(* CoDeSys 2.3.9.48 project: Code_def.pro *)
(* Libraries: standard.lib 2.6.14 10:37:46, Iecsfc.lib 2.6.14 10:37:46, Util.lib 15.3.18 01:28:42, SysLibTime.lib 25.6.18 19:33:14, SysTaskInfo.lib 25.6.18 19:33:14, Syslibs\SysLibRtc.lib 25.6.18 19:33:14, SysLibMem.lib 25.6.18 19:33:14, SYSLIBCALLBACK.LIB 25.6.18 19:33:14, BusDiag.LIB 25.6.18 19:33:14, SysExt_AC500_V10.lib 25.6.18 19:33:14, SysInt_AC500_V10.LIB 25.6.18 19:33:14, MODBUS_AC500_V10.lib 25.6.18 19:33:14 *)

(* PLC configuration (modules and I/O channels)
CPU parameters [AC500_CPU] node 0, in %IB0 out %QB0 {AutoRunType = On; ErrLEDType = On; CheckBatteryType = Off; OutputsInStopType = Off in hardware and online; StopErrorClassType = E2; WarmstartOnFK2Type = Off; FloatingPointExceptionType = E2 failure; IOSimulationModeType = Off; NumberRetainSegmentsType = 8; StartRetainM0Type = 0; EndRetainM0Type = 0; StartRetainM1Type = 0; EndRetainM1Type = 0; StartRetainM2Type = 0; EndRetainM2Type = 0; StartRetainM3Type = 0; EndRetainM3Type = 0; StartRetainM4Type = 0; EndRetainM4Type = 0; StartRetainM5Type = 0; EndRetainM5Type = 0; StartRetainM6Type = 0; EndRetainM6Type = 0; StartRetainM7Type = 0; EndRetainM7Type = 0}
AT %IW0 [WordInputNoSpace] Input 0-15
AT %IB0 [ByteInputNoSpace] Input 0-7
CabStop AT %IX0.0 [BoolInput] Input 0
CabCallP3 AT %IX0.1 [BoolInput] Input 1
CabCallP2 AT %IX0.2 [BoolInput] Input 2
CabCallP1 AT %IX0.3 [BoolInput] Input 3
CabCallP0 AT %IX0.4 [BoolInput] Input 4
CabObstacle AT %IX0.5 [BoolInput] Input 5
Floor3DwBt AT %IX0.6 [BoolInput] Input 6
Floor3DoorClosed AT %IX0.7 [BoolInput] Input 7
AT %IB1 [ByteInputNoSpace] Input 8-15
Floor3DoorOpened AT %IX1.0 [BoolInput] Input 8
Floor3CabPresence AT %IX1.1 [BoolInput] Input 9
Floor2UpBt AT %IX1.2 [BoolInput] Input 10
Floor2DwBt AT %IX1.3 [BoolInput] Input 11
Floor2DoorClosed AT %IX1.4 [BoolInput] Input 12
Floor2DoorOpened AT %IX1.5 [BoolInput] Input 13
Floor2CabPresence AT %IX1.6 [BoolInput] Input 14
Floor1UpBt AT %IX1.7 [BoolInput] Input 15
AT %IW1 [WordInputNoSpace] Input 16-31
AT %IB2 [ByteInputNoSpace] Input 16-23
AT %IX2.0 [BoolInput] Input 16
AT %IX2.1 [BoolInput] Input 17
AT %IX2.2 [BoolInput] Input 18
AT %IX2.3 [BoolInput] Input 19
AT %IX2.4 [BoolInput] Input 20
AT %IX2.5 [BoolInput] Input 21
AT %IX2.6 [BoolInput] Input 22
AT %IX2.7 [BoolInput] Input 23
AT %IB3 [ByteInputNoSpace] Input 24-31
AT %IX3.0 [BoolInput] Input 24
AT %IX3.1 [BoolInput] Input 25
AT %IX3.2 [BoolInput] Input 26
AT %IX3.3 [BoolInput] Input 27
AT %IX3.4 [BoolInput] Input 28
AT %IX3.5 [BoolInput] Input 29
AT %IX3.6 [BoolInput] Input 30
AT %IX3.7 [BoolInput] Input 31
AT %QW0 [WordOutputNoSpace] Output 16-31
AT %QB0 [ByteOutputNoSpace] Output 16-23
CabGoUp AT %QX0.0 [BoolOutput] Output 16
CabGoDown AT %QX0.1 [BoolOutput] Output 17
CabLight AT %QX0.2 [BoolOutput] Output 18
CabLed3 AT %QX0.3 [BoolOutput] Output 19
CabLed2 AT %QX0.4 [BoolOutput] Output 20
CabLed1 AT %QX0.5 [BoolOutput] Output 21
Floor3LedDw AT %QX0.6 [BoolOutput] Output 22
CabLed0 AT %QX0.7 [BoolOutput] Output 23
AT %QB1 [ByteOutputNoSpace] Output 24-31
Floor3DoorClose AT %QX1.0 [BoolOutput] Output 24
Floor3DoorOpen AT %QX1.1 [BoolOutput] Output 25
Floor2LedUp AT %QX1.2 [BoolOutput] Output 26
Floor2LedDw AT %QX1.3 [BoolOutput] Output 27
Floor2DoorClose AT %QX1.4 [BoolOutput] Output 28
Floor2DoorOpen AT %QX1.5 [BoolOutput] Output 29
Floor1LedDw AT %QX1.6 [BoolOutput] Output 30
Floor1LedUp AT %QX1.7 [BoolOutput] Output 31
Fast counter [Module_2FastCounter] node 3, in %IB4 out %QB2
  AT %ID1 [DWordInput] Istwert/Actual value 1
  AT %ID2 [DWordInput] Istwert/Actual value 2
  AT %IB12 [ByteInputNoBits] Statusbyte/State byte 1
  AT %IB13 [ByteInputNoBits] Statusbyte/State byte 2
  AT %QD1 [DWordOutput] Startwert/Start value 1
  AT %QD2 [DWordOutput] Endwert/End value 1
  AT %QD3 [DWordOutput] Startwert/Start value 2
  AT %QD4 [DWordOutput] Endwert/End value 2
  AT %QB20 [ByteOutputNoBits] Steuerbyte/Control byte 1
  AT %QB21 [ByteOutputNoBits] Steuerbyte/Control byte 2
AT %IW7 [WordInputNoSpace] Input 0-15
AT %IB14 [ByteInputNoSpace] Input 0-7
Floor1DwBt AT %IX14.0 [BoolInput] Input 0
Floor1DoorClosed AT %IX14.1 [BoolInput] Input 1
Floor1DoorOpened AT %IX14.2 [BoolInput] Input 2
Floor1CabPresence AT %IX14.3 [BoolInput] Input 3
Floor0UpBt AT %IX14.4 [BoolInput] Input 4
Floor0DoorClosed AT %IX14.5 [BoolInput] Input 5
Floor0DoorOpened AT %IX14.6 [BoolInput] Input 6
Floor0CabPresence AT %IX14.7 [BoolInput] Input 7
AT %IB15 [ByteInputNoSpace] Input 8-15
AT %IX15.0 [BoolInput] Input 8
AT %IX15.1 [BoolInput] Input 9
AT %IX15.2 [BoolInput] Input 10
AT %IX15.3 [BoolInput] Input 11
AT %IX15.4 [BoolInput] Input 12
AT %IX15.5 [BoolInput] Input 13
AT %IX15.6 [BoolInput] Input 14
AT %IX15.7 [BoolInput] Input 15
AT %IW8 [WordInputNoSpace] Input 16-31
AT %IB16 [ByteInputNoSpace] Input 16-23
AT %IX16.0 [BoolInput] Input 16
AT %IX16.1 [BoolInput] Input 17
AT %IX16.2 [BoolInput] Input 18
AT %IX16.3 [BoolInput] Input 19
AT %IX16.4 [BoolInput] Input 20
AT %IX16.5 [BoolInput] Input 21
AT %IX16.6 [BoolInput] Input 22
AT %IX16.7 [BoolInput] Input 23
AT %IB17 [ByteInputNoSpace] Input 24-31
AT %IX17.0 [BoolInput] Input 24
AT %IX17.1 [BoolInput] Input 25
AT %IX17.2 [BoolInput] Input 26
AT %IX17.3 [BoolInput] Input 27
AT %IX17.4 [BoolInput] Input 28
AT %IX17.5 [BoolInput] Input 29
AT %IX17.6 [BoolInput] Input 30
AT %IX17.7 [BoolInput] Input 31
AT %QW11 [WordOutputNoSpace] Output 16-31
AT %QB22 [ByteOutputNoSpace] Output 16-23
Floor1DoorClose AT %QX22.0 [BoolOutput] Output 16
Floor1DoorOpen AT %QX22.1 [BoolOutput] Output 17
Floor0LedUp AT %QX22.2 [BoolOutput] Output 18
Floor0DoorClose AT %QX22.3 [BoolOutput] Output 19
Floor0DoorOpen AT %QX22.4 [BoolOutput] Output 20
AT %QX22.5 [BoolOutput] Output 21
AT %QX22.6 [BoolOutput] Output 22
AT %QX22.7 [BoolOutput] Output 23
AT %QB23 [ByteOutputNoSpace] Output 24-31
AT %QX23.0 [BoolOutput] Output 24
AT %QX23.1 [BoolOutput] Output 25
AT %QX23.2 [BoolOutput] Output 26
AT %QX23.3 [BoolOutput] Output 27
AT %QX23.4 [BoolOutput] Output 28
AT %QX23.5 [BoolOutput] Output 29
AT %QX23.6 [BoolOutput] Output 30
AT %QX23.7 [BoolOutput] Output 31
Fast counter [Module_2FastCounter] node 3, in %IB18 out %QB24
  AT %ID5 [DWordInput] Istwert/Actual value 1
  AT %ID6 [DWordInput] Istwert/Actual value 2
  AT %IB28 [ByteInputNoBits] Statusbyte/State byte 1
  AT %IB29 [ByteInputNoBits] Statusbyte/State byte 2
  AT %QD6 [DWordOutput] Startwert/Start value 1
  AT %QD7 [DWordOutput] Endwert/End value 1
  AT %QD8 [DWordOutput] Startwert/Start value 2
  AT %QD9 [DWordOutput] Endwert/End value 2
  AT %QB40 [ByteOutputNoBits] Steuerbyte/Control byte 1
  AT %QB41 [ByteOutputNoBits] Steuerbyte/Control byte 2
COM1 - MODBUS [AC500_COM1_MODBUS] node 0, in %IB1000 out %QB1000 {COMEnableLoginType = Disabled; COMRTSctrlType = telegram; COMTLSType = 0; COMCDLYType = 0; COMCharTimeoutType = 0; COMTelEndSelType = character timeout; COMTelEndValCharType = 16#00; COMTelEndValWertType = 3; COMChecksumType = CRC16; COMHandshakeType = none; COMBaudType = 19200; COMParityType = none; COMDataBitType = 8; COMStopBitType = 1; COMOperatingModeType = Slave; COMAdressType = 1; COMDisableWriteStartSeg0Type = 0; COMDisableWriteEndSeg0Type = 0; COMDisableReadStartSeg0Type = 0; COMDisableReadEndSeg0Type = 0; COMDisableWriteStartSeg1Type = 0; COMDisableWriteEndSeg1Type = 0; COMDisableReadStartSeg1Type = 0; COMDisableReadEndSeg1Type = 0}
COM2 - Online access [AC500_COM2_Programming] node 1, in %IB2000 out %QB2000 {COMEnableLoginType = Disabled; COMRTSctrlType = telegram; COMTLSType = 0; COMCDLYType = 0; COMCharTimeoutType = 0; COMTelEndSelType = none; COMTelEndValCharType = 16#00; COMTelEndValWertType = 0; COMChecksumType = none; COMHandshakeType = none; COMBaudType = 19200; COMParityType = none; COMDataBitType = 8; COMStopBitType = 1}
FBP - none [AC500_FBP_None] node 2, in %IB3000 out %QB3000
Couplers [AC500_Int_Empty] node 3, in %IB0.0 out %QB0.0
  Internal - none [AC500_IntEmpty] node 0, in %IB4096 out %QB4096 {RunConfigFaultType = No; MaxWaitRunType = 3000; MinUpdateTimeType = 10; ReserveWord0Type = 0; ReserveWord1Type = 0; ReserveWord2Type = 0}
*)

(* Task configuration *)
TASK NewTask (PRIORITY := 10, INTERVAL := T#1ms);
	Main();
END_TASK

(* Global variable list: Global_Variables *)
VAR_GLOBAL
	N: INT:= 6;						(*==============================================================*)
	CabCall: ARRAY [0..5] OF INT;  (*==============================================================*)
	Cabin: CabinDef;
	CallFloor0: BOOL := FALSE;
	CallFloor1: BOOL := FALSE;
	CallFloor2: BOOL := FALSE;
	CallFloor3: BOOL := FALSE;
	Close0 AT %MX0.1.5: BOOL :=FALSE;
	Close1 AT %MX0.1.6: BOOL :=FALSE;
	Close2 AT %MX0.1.7: BOOL :=FALSE;
	Close3 AT %MX0.1.0: BOOL :=FALSE;
	CurrentFloor: UINT;
	DesiredFloor AT %MW0.50: INT;
	Displacement: INT := 450;
	Door0:	INT :=0;
	Door1: INT :=0;
	Door2: INT :=0;
	Door3: INT :=0;
	Door : ARRAY [0..5] OF INT;		(*==============================================================*)
	DoorClosed0 AT %MX0.6.0: BOOL;
	DoorClosed1 AT %MX0.6.2: BOOL;
	DoorClosed2 AT %MX0.6.4: BOOL;
	DoorClosed3 AT %MX0.6.6: BOOL;
	DoorOpened0 AT %MX0.6.1: BOOL;
	DoorOpened1 AT %MX0.6.3: BOOL;
	DoorOpened2 AT %MX0.6.5: BOOL;
	DoorOpened3 AT %MX0.6.7: BOOL;
	DwCall: ARRAY [0..5] OF INT;		(*==============================================================*)
	DwCall1 AT %MW0.61: INT;
	DwCall2 AT %MW0.62: INT;
	DwCall3 AT %MW0.63: INT;
	DwCall4 AT %MW0.64: INT;
	EndMovement: BOOL;
	EndMovementObstacle: BOOL := FALSE;
	EndOpening: BOOL;
	EndOpeningObstacle: BOOL := FALSE;
	Error AT %MW0.4: INT := 0;
	ErrorOpeningDoor: ARRAY [0..5] OF BOOL;	(*==============================================================*)
	ErrorClosingDoor: ARRAY [0..5] OF BOOL;(*==============================================================*)
	Floor: ARRAY[0..5] OF FloorDef;  			(*==============================================================*)
	FloorIndicator AT %MW0.2: UINT;
	GoDw AT %MX0.0.3: BOOL :=FALSE;
	GoUp AT %MX0.0.2: BOOL :=FALSE;
	Init AT %MX0.0.0: BOOL := FALSE;
	IntCall1 AT %MW0.53: INT;
	IntCall2 AT %MW0.54: INT;
	IntCall3 AT %MW0.55: INT;
	IntCall4 AT %MW0.56: INT;

	IntermittingLightOFF: BOOL;
	IntermittingLightON: BOOL;
	isBetween: ARRAY [0..5] OF BOOL;  (*==============================================================*)
	LimitWeight AT %MW0.52: INT:=320;
	Man AT %MX0.0.1:  BOOL := FALSE;

	MovedDw: BOOL;
	MovedUp: BOOL;
	MovingDw: BOOL;
	MovingUp: BOOL;
	Multiple: BOOL := FALSE;
	ObstacleCase: BOOL := FALSE;
	ObstacleOccurred: BOOL := FALSE;
	Open0 AT %MX0.1.1: BOOL := FALSE;
	Open1 AT %MX0.1.2: BOOL := FALSE;
	Open2 AT %MX0.1.3: BOOL := FALSE;
	Open3 AT %MX0.1.4: BOOL := FALSE;
	Optimized: BOOL := FALSE;
	PreviousLogic: INT;
	Queue: ARRAY [0..5] OF INT;			(*==============================================================*)
	Queue1 AT %MW0.65: INT;
	Queue2 AT %MW0.66: INT;
	Queue3 AT %MW0.67: INT;
	Queue4 AT %MW0.68: INT;
	ReadyToDelete: BOOL;
	ReadyToMove: BOOL;
	Single: BOOL := FALSE;
	StartClose: BOOL;
	StartCloseAfterObstacle: BOOL;
	StopOccurred: BOOL := FALSE;
	TimerCabLightOFF: BOOL;
	TimerDelete: BOOL;
	TimerDoor: BOOL;
	TimerDoorAfterObstacle: BOOL;
	TimerErrorCabin: BOOL := FALSE;
	TimerErrorOpeningDoor: ARRAY [0..5] OF BOOL:= FALSE; (*==============================================================*)
	TimerErrorClosingDoor: ARRAY [0..5] OF BOOL:= FALSE;(*==============================================================*)
	TimerIntermittingLightOFF: BOOL;
	TimerIntermittingLightON: BOOL;
	TimerReOpening: BOOL;
	UpCall: ARRAY [0..5] OF INT;(*==============================================================*)
	UpCall1 AT %MW0.57: INT;
	UpCall2 AT %MW0.58: INT;
	UpCall3 AT %MW0.59: INT;
	UpCall4 AT %MW0.60: INT;
	Weight AT %MW0.51: INT;
END_VAR

(* Data type *)
TYPE CabinDef :
STRUCT

	Call:ARRAY [0..5] OF BOOL;	(*==============================================================*)
	GoUp: BOOL;
	GoDown: BOOL;
	Light: BOOL;
	Obstacle: BOOL;
	Stop: BOOL;
	ErrorCabin: BOOL;

END_STRUCT
END_TYPE

(* Data type *)
TYPE FloorDef :
STRUCT

	DoorClose: BOOL;
	DoorOpen: BOOL;
	DoorOpened: BOOL;
	DoorClosed: BOOL;
	CabPresence: BOOL;
	CallUp: BOOL;
	CallDw: BOOL;
	CabLed: BOOL;
	LedUp: BOOL;
	LedDw: BOOL;

END_STRUCT
END_TYPE

(* POU Main, ST *)
PROGRAM Main
VAR
	CabLightOFF: BOOL;
	i: INT;
	Logic AT %MW0.5: INT := 3;
	OverWeight: BOOL;
	Sim: BOOL := FALSE;
	TimerStop: BOOL;
	TON_CabLightOFF: TON;
	TON_Delete: TON;
	TON_Door: TON;
	TON_ErrorCabin: TON;
	TON_ErrorOpeningDoor: ARRAY[0..5] OF TON;   (*==============================================================*)
	TON_ErrorClosingDoor: ARRAY[0..5] OF TON;	(*==============================================================*)
	TON_Obstacle: TON;
	TON_ReOpening: TON;
	TON_StopLightOFF: TON;
	TON_StopLightON: TON;
	CountDoorClosed: INT;
	CountErrorClosingDoor : INT;
	CountErrorOpeningDoor: INT;
END_VAR
IF (Sim = FALSE) THEN
	ASS_INPUT;
	(*HMI;*)
ELSE
	SIMULATION_INPUT;
END_IF

IF (Man = TRUE) THEN
	(*MANUAL;*)
	;
ELSE

(*-------------------------------------------------------initialization----------------------------------------------------*)
	IF( Init = FALSE) THEN
		Init := Initialize();
	ELSE

		TON_StopLightOFF(IN:= TimerIntermittingLightOFF, PT:= T#1s, Q=> IntermittingLightOFF);
		TON_StopLightON(IN:= TimerIntermittingLightON, PT:= T#1s, Q=> IntermittingLightON);

		(*CountDoorClosed = N if all doors are closed 		    *)
		(*					   < N if at least one door is opened *)
		(*CountErrorClosingDoor = N if no error during closing door*)
		(*							 <N ia there is an error during closing door*)
		(*CountErrorOpeningDoor = N if no error during opening door*)
		(*							 <N ia there is an error during opening door*)
		CountDoorClosed := 0;
		CountErrorClosingDoor := 0;
		CountErrorOpeningDoor  := 0;

		FOR i := 0 TO N-1 DO
			IF (Floor[i].DoorClosed = TRUE) THEN
				CountDoorClosed := CountDoorClosed +1;
			END_IF
			IF (ErrorClosingDoor[i] = FALSE) THEN
				CountErrorClosingDoor := CountErrorClosingDoor + 1;
			END_IF
			IF (ErrorOpeningDoor[i] = FALSE) THEN
				CountErrorOpeningDoor := CountErrorOpeningDoor + 1;
			END_IF
		END_FOR


		IF (CountDoorClosed < N AND Weight > LimitWeight) THEN
			OverWeight := TRUE;
		ELSE
			OverWeight:= FALSE;
		END_IF

		IF (Cabin.ErrorCabin = FALSE AND CountErrorClosingDoor = N AND CountErrorOpeningDoor = N  AND OverWeight = FALSE) THEN
			(*----------------------------------------------------Timers Definition-----------------------------------------------*)

			TON_CabLightOFF(IN:= TimerCabLightOFF, PT:= T#5s, Q=> CabLightOFF);
			TON_Delete(IN:= TimerDelete, PT:= T#3s, Q=> ReadyToDelete);
			TON_Door(IN:= TimerDoor, PT:= T#5s, Q=> StartClose);
			TON_ErrorCabin (IN:= TimerErrorCabin, PT:= T#10s, Q=> Cabin.ErrorCabin);
			TON_Obstacle(IN:= TimerDoorAfterObstacle, PT:= T#2s, Q=> StartCloseAfterObstacle);
			TON_ReOpening(IN:= TimerReOpening, PT:= T#3s, Q=> ReadyToMove);

			FOR i := 0 TO N-1 DO
				TON_ErrorClosingDoor[i](IN:= TimerErrorClosingDoor[i], PT:= T#10s, Q=> ErrorClosingDoor[i]);
				TON_ErrorOpeningDoor[i](IN:= TimerErrorOpeningDoor[i], PT:= T#10s, Q=> ErrorOpeningDoor[i]);
			END_FOR

			(*
			TON_ErrorClosingDoor0 (IN:= TimerErrorClosingDoor0, PT:= T#10s, Q=> ErrorClosingDoor0);
			TON_ErrorClosingDoor1 (IN:= TimerErrorClosingDoor1, PT:= T#10s, Q=> ErrorClosingDoor1);
			TON_ErrorClosingDoor2 (IN:= TimerErrorClosingDoor2, PT:= T#10s, Q=> ErrorClosingDoor2);
			TON_ErrorClosingDoor3 (IN:= TimerErrorClosingDoor3, PT:= T#10s, Q=> ErrorClosingDoor3);
			TON_ErrorOpeningDoor0 (IN:= TimerErrorOpeningDoor0, PT:= T#10s, Q=> ErrorOpeningDoor0);
			TON_ErrorOpeningDoor1 (IN:= TimerErrorOpeningDoor1, PT:= T#10s, Q=> ErrorOpeningDoor1);
			TON_ErrorOpeningDoor2 (IN:= TimerErrorOpeningDoor2, PT:= T#10s, Q=> ErrorOpeningDoor2);
			TON_ErrorOpeningDoor3 (IN:= TimerErrorOpeningDoor3, PT:= T#10s, Q=> ErrorOpeningDoor3);*)


			(*---------------------------------------------------Main Program----------------------------------------------------*)

			IF(CountDoorClosed = N AND Cabin.GoDown = FALSE AND Cabin.GoUp = FALSE) THEN
				TimerReOpening := TRUE;
				TimerDelete := TRUE;
			END_IF

			IF(CountDoorClosed = N AND Cabin.GoDown = FALSE AND Cabin.GoUp = FALSE AND (EndMovement = TRUE OR DesiredFloor = -1)) THEN
				Logic_Choice(Logic);
			END_IF

			IF(ReadyToMove = TRUE) THEN
				TimerCabLightOFF := TRUE;
			END_IF

			IF(CountDoorClosed < N) THEN
				TimerReOpening := FALSE;
				TimerDelete := FALSE;
			END_IF

			Case_Division();
			Define_Current_Floor(StopOccurred);
			IF (Single = TRUE) THEN
				Define_Desired_Floor();
			ELSIF (Multiple = TRUE) THEN
				Add_To_Queue();
				DesiredFloor := Queue[0];
			ELSIF (Optimized = TRUE) THEN
				Add_To_Calls();
				IF (DesiredFloor <> CurrentFloor) THEN
					Manage_Calls();
				END_IF
			END_IF

			(*-------------------------------------------------------No Obstacle---------------------------------------------------*)
			IF(ObstacleCase = FALSE) THEN
				IF (ReadyToMove = TRUE) THEN
					Movement_Management();
				END_IF
				Doors_Management_No_Obstacle();
			(*---------------------------------------------------------Obstacle------------------------------------------------------*)
			ELSIF ((Cabin.Obstacle = TRUE OR ObstacleCase = TRUE) AND Cabin.GoDown = FALSE AND Cabin.GoUp = FALSE AND StopOccurred = FALSE) THEN
				Obstacle_Function();
				Doors_Management_Obstacle();
			END_IF
			(*----------------------------------------------------------------------------------------------------------------------------*)

			IF (CabLightOFF = TRUE) THEN
				Cabin.Light := FALSE;
			ELSE
				Cabin.Light := TRUE;
			END_IF

		ELSIF (OverWeight = TRUE AND Cabin.GoDown = FALSE AND Cabin.GoUp = FALSE) THEN
			Open_Door(CurrentFloor);
			Floor[CurrentFloor].DoorClose := FALSE;
			FOR i := 0 TO N-1 DO
				TimerErrorOpeningDoor[i] := FALSE;
				TimerErrorClosingDoor[i] := FALSE;
			END_FOR

			IF (TimerIntermittingLightOFF = FALSE) THEN
				TimerIntermittingLightON := TRUE;
			END_IF

			IF(IntermittingLightON = TRUE) THEN
				Floor[CurrentFloor].CabLed := TRUE;
				TimerIntermittingLightOFF := TRUE;
				TimerIntermittingLightON := FALSE;
			END_IF

			IF(IntermittingLightOFF = TRUE) THEN
				Floor[CurrentFloor].CabLed := FALSE;
				TimerIntermittingLightON := TRUE;
				TimerIntermittingLightOFF := FALSE;
			END_IF
		ELSE
			Error_Management();
		END_IF

	END_IF

END_IF

 (*---------------------------------------------------------------------------------------------------------------------------*)

ASS_OUTPUT;
END_PROGRAM

(* POU ASS_INPUT, ST *)
PROGRAM ASS_INPUT
VAR
	i : INT;
END_VAR
(*Floor 0 Assignment*)
Floor[0].CabPresence	:= Floor0CabPresence;
Floor[0].DoorClosed		:= Floor0DoorClosed;
Floor[0].DoorOpened		:= Floor0DoorOpened;
Floor[0].CallUp			:= Floor0UpBt;

(*Floor 1 Assignment*)
Floor[1].CabPresence	:= Floor1CabPresence;
Floor[1].DoorClosed		:= Floor1DoorClosed;
Floor[1].DoorOpened		:= Floor1DoorOpened;
Floor[1].CallUp			:= Floor1UpBt;
Floor[1].CallDw			:= Floor1DwBt;

(*Floor 2 Assignment*)
Floor[2].CabPresence	:= Floor2CabPresence;
Floor[2].DoorClosed		:= Floor2DoorClosed;
Floor[2].DoorOpened		:= Floor2DoorOpened;
Floor[2].CallUp			:= Floor2UpBt;
Floor[2].CallDw 			:= Floor2DwBt;

(*Floor 3 Assignment*)
Floor[3].CabPresence	:= Floor3CabPresence;
Floor[3].DoorClosed		:= Floor3DoorClosed;
Floor[3].DoorOpened		:= Floor3DoorOpened;
Floor[3].CallDw 			:= Floor3DwBt;

(*Cabin Assignment*)
Cabin.Call[0]				:= CabCallP0;
Cabin.Call[1]				:= CabCallP1;
Cabin.Call[2]				:= CabCallP2;
Cabin.Call[3]				:= CabCallP3;
Cabin.Obstacle			:= CabObstacle;
Cabin.Stop				:= CabStop;
END_PROGRAM

(* POU SIMULATION_INPUT, ST *)
PROGRAM SIMULATION_INPUT
VAR
END_VAR
(*Floor 0 Assignment*)
IF (Displacement = 450) THEN
	Floor[0].CabPresence	:= TRUE;
ELSIF (Displacement < 445) THEN
	Floor[0].CabPresence	:= FALSE;
END_IF
IF (Door0 = 0) THEN
	Floor[0].DoorClosed		:= TRUE;
ELSE
	Floor[0].DoorClosed		:= FALSE;
END_IF
IF (Door0 = 110) THEN
	Floor[0].DoorOpened		:= TRUE;
ELSE
	Floor[0].DoorOpened		:= FALSE;
END_IF
Floor[0].CallUp				:= Floor0UpBt;

(*Floor 1 Assignment*)
IF (Displacement = 300) THEN
	Floor[1].CabPresence	:= TRUE;
ELSIF (Displacement < 295 OR Displacement > 305) THEN
	Floor[1].CabPresence	:= FALSE;
END_IF
IF (Door1 = 0) THEN
	Floor[1].DoorClosed		:= TRUE;
ELSE
	Floor[1].DoorClosed		:= FALSE;
END_IF
IF (Door1 = 110) THEN
	Floor[1].DoorOpened		:= TRUE;
ELSE
	Floor[1].DoorOpened		:= FALSE;
END_IF
Floor[1].CallUp				:= Floor1UpBt;
Floor[1].CallDw				:= Floor1DwBt;

(*Floor 2 Assignment*)
IF (Displacement = 150) THEN
	Floor[2].CabPresence	:= TRUE;
ELSIF (Displacement < 145 OR Displacement > 155) THEN
	Floor[2].CabPresence	:= FALSE;
END_IF
IF (Door2 = 0) THEN
	Floor[2].DoorClosed		:= TRUE;
ELSE
	Floor[2].DoorClosed		:= FALSE;
END_IF
IF (Door2 = 110) THEN
	Floor[2].DoorOpened		:= TRUE;
ELSE
	Floor[2].DoorOpened		:= FALSE;
END_IF
Floor[2].CallUp				:= Floor2UpBt;
Floor[2].CallDw 				:= Floor2DwBt;

(*Floor 3 Assignment*)
IF (Displacement = 0) THEN
	Floor[3].CabPresence	:= TRUE;
ELSIF (Displacement > 5) THEN
	Floor[3].CabPresence	:= FALSE;
END_IF
IF (Door3 = 0) THEN
	Floor[3].DoorClosed		:= TRUE;
ELSE
	Floor[3].DoorClosed		:= FALSE;
END_IF
IF (Door3 = 110) THEN
	Floor[3].DoorOpened		:= TRUE;
ELSE
	Floor[3].DoorOpened		:= FALSE;
END_IF
Floor[3].CallDw 				:= Floor3DwBt;

(*Cabin Assignment*)
Cabin.Call[0]					:= CabCallP0;
Cabin.Call[1]					:= CabCallP1;
Cabin.Call[2]					:= CabCallP2;
Cabin.Call[3]					:= CabCallP3;
Cabin.Obstacle				:= CabObstacle;
Cabin.Stop					:= CabStop;
END_PROGRAM

(* POU Initialize, ST *)
FUNCTION Initialize: BOOL
VAR_INPUT
END_VAR
VAR
	i: INT;
	CountDoorClosed : INT;
END_VAR
FOR i := 0 TO N-1 DO
	(*Reset All Queues *)
	Queue[i] := -1;
	CabCall[i] := -1;
	UpCall[i] := -1;
	DwCall[i] := -1;
	(*Turn Off All Lights*)
	Floor[i].CabLed := FALSE;
	Floor[i].LedUp := FALSE;
	Floor[i].LedDw := FALSE;
END_FOR


FOR i := 0 TO N-1 DO
	IF(Floor[i].DoorClosed = FALSE) THEN
		Floor[i].DoorClose := TRUE;
	ELSE
		Floor[i].DoorClose := FALSE;
	END_IF
END_FOR

(*Door Floor  0*)
IF(Floor[0].DoorClosed = FALSE) THEN
	Door0 := Door0 - 1;
END_IF

(*Door Floor 1*)
IF(Floor[1].DoorClosed = FALSE) THEN
	Door1 := Door1 - 1;
END_IF

(*Door Floor 2*)
IF(Floor[2].DoorClosed = FALSE) THEN
	Door2 := Door2 - 1;
END_IF

(*Door Floor 3*)
IF(Floor[3].DoorClosed = FALSE) THEN
	Door3 := Door3 - 1;
END_IF

CountDoorClosed := 0;
FOR i := 0 TO N-1 DO
	IF (Floor[i].DoorClosed = TRUE) THEN
		CountDoorClosed := CountDoorClosed +1;
	END_IF
END_FOR

(*Cabin Floor 0*)
IF (Floor[0].CabPresence = FALSE AND CountDoorClosed = N) THEN
	Cabin.GoDown := TRUE;
	Displacement := Displacement +1;
ELSE
	Cabin.GoDown := FALSE;
END_IF

(*Variable Initialization*)
IF (Floor[0].CabPresence = TRUE AND CountDoorClosed = N) THEN
	Cabin.ErrorCabin := FALSE;
	DesiredFloor := -1;
	EndMovement := TRUE;
	EndOpening:=FALSE;
	FOR i := 0 TO N-1 DO
		ErrorClosingDoor[i] := FALSE;
		ErrorOpeningDoor[i] := FALSE;
		TimerErrorClosingDoor[i] := FALSE;
		TimerErrorOpeningDoor[i] := FALSE;
	END_FOR

	Initialize := TRUE;
	FOR i:= 0 TO N-2 DO
		IsBetween[i] := FALSE;
	END_FOR;
	MovingDw := FALSE;
	MovingUp:= FALSE;
	MovedDw := FALSE;
	MovedUp := FALSE;
	ObstacleCase := FALSE;
	ObstacleOccurred := FALSE;
	StopOccurred := FALSE;
	TimerCabLightOFF := FALSE;
	TimerDelete := TRUE;
	TimerDoor := FALSE;
	TimerDoorAfterObstacle := FALSE;
	TimerErrorCabin := FALSE;
	TimerIntermittingLightOFF := FALSE;
	TimerIntermittingLightON := FALSE;
	TimerReOpening := TRUE;
ELSE
	Initialize := FALSE;
END_IF

(*
Door0 := Door[0];
Door1 := Door[1];
Door2 := Door[2];
Door3 := Door[3];*)
END_FUNCTION

(* POU Logic_Choice, ST *)
FUNCTION Logic_Choice: BOOL
VAR_INPUT
	Logic : INT;
END_VAR
VAR
END_VAR
IF (Logic = 1) THEN
	Single := TRUE;
	Multiple := FALSE;
	Optimized := FALSE;
ELSIF (Logic = 2) THEN
	Single := FALSE;
	Multiple := TRUE;
	Optimized := FALSE;
ELSIF (Logic = 3) THEN
	Single := FALSE;
	Multiple := FALSE;
	Optimized := TRUE;
END_IF

IF (Logic <> PreviousLogic) THEN
	Init := FALSE;
END_IF

PreviousLogic := Logic;
END_FUNCTION

(* POU Case_Division, ST *)
FUNCTION Case_Division: BOOL
VAR_INPUT
END_VAR
VAR
	CountCabPresence : INT;
	i : INT;
END_VAR
CountCabPresence := 0;
FOR i := 0 TO N-1 DO
	IF (Floor[i].CabPresence= FALSE) THEN
		CountCabPresence := CountCabPresence + 1;
	END_IF
END_FOR

IF (Cabin.Stop = TRUE AND CountCabPresence = N) THEN
	StopOccurred := TRUE;
END_IF

IF ((Cabin.Obstacle = TRUE OR ObstacleCase = TRUE) AND Cabin.GoDown = FALSE AND Cabin.GoUp = FALSE AND StopOccurred = FALSE) THEN
	ObstacleCase := TRUE;
ELSE
	ObstacleCase := FALSE;
END_IF
END_FUNCTION

(* POU Define_Current_Floor, ST *)
FUNCTION Define_Current_Floor: BOOL
VAR_INPUT
	StopOccurred: BOOL;
END_VAR
VAR
	i : INT;
END_VAR
FOR i := 0 TO N-1 DO
	IF (Floor[i].CabPresence = TRUE) THEN
		CurrentFloor := i;
		Floor[i].CabLed := TRUE;
	ELSIF (StopOccurred = FALSE) THEN
		Floor[i].CabLed := FALSE;
	END_IF
END_FOR

i := 0;
IF((CurrentFloor = i AND MovingUp = TRUE  AND Floor[i].CabPresence = FALSE) OR (CurrentFloor = i+1 AND MovingDw = TRUE  AND Floor[i+1].CabPresence = FALSE AND IsBetween[i+1] = FALSE)) THEN
	IsBetween[i] := TRUE;
ELSIF (Floor[i].CabPresence = TRUE OR Floor[i+1].CabPresence = TRUE) THEN
	IsBetween[i] := FALSE;
END_IF

FOR i:= 1 TO N-3 DO
	IF((CurrentFloor = i AND MovingUp = TRUE AND Floor[i].CabPresence = FALSE AND IsBetween[i-1] = FALSE) OR (CurrentFloor = i+1 AND MovingDw = TRUE AND Floor[i+1].CabPresence = FALSE AND IsBetween[i+1] = FALSE)) THEN
		IsBetween[i] := TRUE;
	ELSIF (Floor[i].CabPresence = TRUE OR Floor[i+1].CabPresence = TRUE) THEN
		IsBetween[i] := FALSE;
	END_IF
END_FOR

i := N-2;
IF((CurrentFloor = i AND MovingUp = TRUE AND Floor[i].CabPresence = FALSE AND IsBetween[i-1] = FALSE) OR (CurrentFloor = i+1 AND MovingDw = TRUE AND Floor[i+1].CabPresence = FALSE)) THEN
	IsBetween[i] := TRUE;
ELSIF (Floor[i].CabPresence = TRUE OR Floor[i+1].CabPresence = TRUE) THEN
	IsBetween[i] := FALSE;
END_IF
END_FUNCTION

(* POU Define_Desired_Floor, ST *)
FUNCTION Define_Desired_Floor: BOOL
VAR_INPUT
END_VAR
VAR
	i : INT;
END_VAR
IF (DesiredFloor = -1) THEN
	FOR i := 0 TO N-1 DO
		IF (Cabin.Call[i] = TRUE) THEN
			DesiredFloor := i;
		END_IF
		IF (Floor[i].CallUp = TRUE AND i <> N-1) THEN
			DesiredFloor := i;
			Floor[i].LedUp := TRUE;
		END_IF
		IF (Floor[i].CallDw = TRUE AND i <> 0) THEN
			DesiredFloor := i;
			Floor[i].LedDw := TRUE;
		END_IF
	END_FOR
END_IF
END_FUNCTION

(* POU Add_To_Queue, ST *)
FUNCTION Add_To_Queue: BOOL
VAR_INPUT
END_VAR
VAR
	Rec: BOOL := FALSE;
	i: INT;
	j : INT;
	IsPresent: ARRAY [0..5] OF BOOL;(*==============================================================*)
END_VAR
FOR j := 0 TO N-1 DO
	FOR i := 0 TO N-1 DO
		IF (Queue[j] = i) THEN
			IsPresent[i] := TRUE;
		END_IF
	END_FOR
END_FOR

i := 0 ;
IF(Cabin.Call[i] = TRUE OR Floor[i].CallUp = TRUE)  THEN
	IF (Floor[i].CabPresence = TRUE AND ReadyToMove = FALSE  AND IsPresent[i] = FALSE) THEN
		Add_First_To_Queue(i);
	ELSIF (IsPresent[i] = FALSE) THEN
		Add_Last_To_Queue(i);
	END_IF
	IF (Floor[i].CallUp = TRUE)  THEN
		Floor[i].LedUp := TRUE;
	END_IF
END_IF

FOR i := 1 TO N-2 DO
	IF (Cabin.Call[i] = TRUE OR Floor[i].CallUp = TRUE OR Floor[i].CallDw = TRUE) THEN
		IF (Floor[i].CabPresence = TRUE AND ReadyToMove = FALSE AND IsPresent[i] = FALSE) THEN
			Add_First_To_Queue(i);
		ELSIF (IsPresent[i] = FALSE) THEN
			Add_Last_To_Queue(i);
		END_IF
		IF (Floor[i].CallUp = TRUE) THEN
			Floor[i].LedUp := TRUE;
		ELSIF (Floor[i].CallDw = TRUE) THEN
			Floor[i].LedDw := TRUE;
		END_IF
	END_IF
END_FOR

i := N-1;
IF(Cabin.Call[i] = TRUE OR Floor[i].CallDw = TRUE) THEN
	IF (Floor[i].CabPresence = TRUE AND ReadyToMove = FALSE AND IsPresent[i] = FALSE) THEN
		Add_First_To_Queue(i);
	ELSIF (IsPresent[i] = FALSE) THEN
		Add_Last_To_Queue(i);
	END_IF
	IF (Floor[i].CallDw = TRUE) THEN
		Floor[i].LedDw := TRUE;
	END_IF
END_IF
END_FUNCTION

(* POU Add_First_To_Queue, ST *)
FUNCTION Add_First_To_Queue: BOOL
VAR_INPUT
	DesFloor: INT;
END_VAR
VAR
	i: INT;
	Temp1: ARRAY [0..5] OF INT;	(*==============================================================*)
	Temp2: ARRAY [0..5] OF INT;	(*==============================================================*)
END_VAR
Temp1[0] := DesFloor;
Temp2 := Queue;
FOR i := 1 TO N-1 DO
	Temp1[i] := Temp2[i-1];
END_FOR

Queue := Temp1;
END_FUNCTION

(* POU Add_Last_To_Queue, ST *)
FUNCTION Add_Last_To_Queue: BOOL
VAR_INPUT
	DesFloor: INT;
END_VAR
VAR
	Rec: BOOL := FALSE;
	i: INT;
END_VAR
FOR i:= 0 TO N-1 DO
	IF (Queue[i] = -1 AND Rec = FALSE) THEN
		Queue[i] := DesFloor;
		Rec := TRUE;
	END_IF
END_FOR
END_FUNCTION

(* POU Add_To_Calls, ST *)
FUNCTION Add_To_Calls: BOOL
VAR_INPUT
END_VAR
VAR
	i: INT;
	j : INT;
	IsPresent: ARRAY [0..5] OF BOOL;	(*==============================================================*)
	IsPresentUp: ARRAY [0..5] OF BOOL;(*==============================================================*)
	IsPresentDw: ARRAY [0..5] OF BOOL;(*==============================================================*)
END_VAR
FOR j:= 0 TO N-1 DO
	FOR i := 0 TO N-1 DO
		IF (CabCall[j] = i) THEN
			IsPresent[i] := TRUE;
		END_IF

		IF (UpCall[j] = i AND i<> N-1) THEN
			IsPresentUp[i] := TRUE;
		END_IF

		IF (DwCall[j] =i AND i <> 0) THEN
			IsPresentDw[i] := TRUE;
		END_IF
	END_FOR
END_FOR

i:=0;
IF(Cabin.Call[i] = TRUE AND IsPresent[i] = FALSE) THEN
		Add_Last_To_Calls(i,0);
END_IF

IF(Floor[i].CallUp = TRUE AND IsPresentUp[i] = FALSE) THEN
		Add_Last_To_Calls(i,1);
		Floor[i].LedUp := TRUE;
END_IF

FOR i := 1 TO N-2 DO
	IF(Cabin.Call[i] = TRUE AND IsPresent[i] = FALSE) THEN
		Add_Last_To_Calls(i,0);
	END_IF

	IF(Floor[i].CallUp = TRUE AND IsPresentUp[i] = FALSE) THEN
		Add_Last_To_Calls(i,1);
		Floor[i].LedUp := TRUE;
	END_IF

	IF(Floor[i].CallDw = TRUE AND IsPresentDw[i] = FALSE) THEN
		Add_Last_To_Calls(i,2);
		Floor[i].LedDw := TRUE;
	END_IF
END_FOR

i:= N-1;
IF(Cabin.Call[i] = TRUE AND IsPresent[i] = FALSE) THEN
		Add_Last_To_Calls(i,0);
END_IF

IF(Floor[i].CallDw = TRUE AND IsPresentDw[i] = FALSE) THEN
		Add_Last_To_Calls(i,2);
		Floor[i].LedDw := TRUE;
END_IF
END_FUNCTION

(* POU Add_Last_To_Calls, ST *)
FUNCTION Add_Last_To_Calls: BOOL
VAR_INPUT
	DesFloor: INT;
	TargetArray: INT;
END_VAR
VAR
	Rec: BOOL := FALSE;
	i: INT;
END_VAR
CASE TargetArray OF
0:	FOR i := 0 TO N-1 DO
		IF (CabCall[i] = -1 AND Rec = FALSE) THEN
			CabCall[i] := DesFloor;
			Rec :=TRUE;
		END_IF
	END_FOR
1:	FOR i:= 0 TO N-1 DO
		IF (UpCall[i] = -1 AND Rec = FALSE) THEN
			UpCall[i] := DesFloor;
			Rec :=TRUE;
		END_IF
	END_FOR
2:	FOR i:= 0 TO N-1 DO
		IF (DwCall[i] = -1 AND Rec = FALSE) THEN
			DwCall[i] := DesFloor;
			Rec :=TRUE;
		END_IF
	END_FOR
END_CASE
END_FUNCTION

(* POU Manage_Calls, ST *)
FUNCTION Manage_Calls: BOOL
VAR_INPUT
END_VAR
VAR
	i: INT;
	Temp: INT;
	Count: INT := 0;
END_VAR
IF ((MovedUp = TRUE OR MovedDw = FALSE) AND StopOccurred = FALSE) THEN
	Temp := 100;
	FOR i := 0 TO N-1 DO
		IF (CabCall[i] > CurrentFloor AND CabCall[i] < Temp AND CabCall[i] <> -1) THEN
			Temp := CabCall[i];
		END_IF
		IF (UpCall[i] > CurrentFloor AND UpCall[i] < Temp AND UpCall[i] <> -1) THEN
			Temp := UpCall[i];
		END_IF
	END_FOR
	IF (Temp = 100) THEN
		Temp := -100;
		FOR i := 0 TO N-1 DO
			IF (DwCall[i] > Temp AND DwCall[i] <> -1) THEN
				Temp := DwCall[i];
			END_IF
		END_FOR
	END_IF
	FOR i := 0 TO N-1 DO
		IF (CabCall[0] = -1 AND DwCall[0] = -1 AND UpCall[i] < CurrentFloor) THEN
			Count := Count +1;
		END_IF
	END_FOR
	IF (Count = N) THEN
		Temp := 100;
		FOR i := 0 TO N-1 DO
			IF (UpCall[i] < Temp AND UpCall[i] <> -1) THEN
				Temp := UpCall[i];
			END_IF
		END_FOR
	END_IF
	IF (Temp <> 100 AND Temp <> -100) THEN
		DesiredFloor := Temp;
		IF (DesiredFloor < CurrentFloor) THEN
			MovedUp := FALSE;
		END_IF
	ELSE
		MovedUp := FALSE;
	END_IF
END_IF

IF ((MovedDw = TRUE OR MovedUp = FALSE) AND StopOccurred = FALSE) THEN
	Temp := -100;
	FOR i := 0 TO N-1 DO
		IF(CabCall[i] < CurrentFloor AND CabCall[i] > Temp AND CabCall[i] <> -1) THEN
			Temp := CabCall[i];
		END_IF
		IF(DwCall[i] < CurrentFloor AND DwCall[i] > Temp AND DwCall[i] <> -1) THEN
			Temp := DwCall[i];
		END_IF
	END_FOR
	IF (Temp = -100) THEN
		Temp := 100;
		FOR i := 0 TO N-1 DO
			IF(UpCall[i] < Temp AND UpCall[i] <> -1) THEN
				Temp := UpCall[i];
			END_IF
		END_FOR
	END_IF
	FOR i := 0 TO N-1 DO
		IF (CabCall[0] = -1 AND UpCall[0] = -1 AND DwCall[i] > CurrentFloor) THEN
			Count := Count +1;
		END_IF
	END_FOR
	IF (Count = N) THEN
		Temp := -100;
		FOR i := 0 TO N-1 DO
			IF (DwCall[i] > Temp AND DwCall[i] <> -1) THEN
				Temp := DwCall[i];
			END_IF
		END_FOR
	END_IF
	IF (Temp <> 100 AND Temp <> -100) THEN
		DesiredFloor := Temp;
		IF (DesiredFloor > CurrentFloor) THEN
			MovedDw := FALSE;
		END_IF
	ELSE
		MovedDw := FALSE;
	END_IF
END_IF

IF (StopOccurred = TRUE AND DesiredFloor = -1) THEN
	i:= 0;
	IF (CabCall[0] = i OR UpCall[0] = i) THEN
		DesiredFloor := 0;
	END_IF
	FOR i:= 1 TO N-2 DO
		IF (CabCall[0] = i OR UpCall[0] = i OR DwCall[0] = i) THEN
			DesiredFloor := i;
		END_IF
	END_FOR
	i:= N-1;
	IF (CabCall[0] = i OR DwCall[0] = i) THEN
		DesiredFloor := i;
	END_IF
END_IF
END_FUNCTION

(* POU Movement_Management, ST *)
FUNCTION Movement_Management: BOOL
VAR_INPUT
END_VAR
VAR
	i:INT;
	CountCabPresence : INT ;
END_VAR
CountCabPresence := 0;
FOR i := 0 TO N-1 DO
	IF (Floor[i].CabPresence = FALSE) THEN
		CountCabPresence := CountCabPresence +1;
	END_IF
END_FOR

IF (Cabin.Stop = TRUE AND CountCabPresence = N) THEN
	DesiredFloor := -1;
	Cabin.GoDown := FALSE;
	Cabin.GoUp := FALSE;
	StopOccurred := TRUE;
	TimerIntermittingLightON := TRUE;
	TimerIntermittingLightOFF := FALSE;
	TimerErrorCabin := FALSE;
	FOR i:= 0 TO N-1 DO
		IF (i<> N-1) THEN
			Floor[i].LedUp := FALSE;
		END_IF
		IF (i<> 0) THEN
			Floor[i].LedDw := FALSE;
		END_IF
	END_FOR
	IF (Multiple = TRUE OR Optimized = TRUE) THEN
		Delete_All_Queue();
	END_IF
END_IF

IF(IntermittingLightON = TRUE AND StopOccurred = TRUE AND DesiredFloor = -1) THEN
	FOR i:= 0 TO N-1 DO
		Floor[i].CabLed := TRUE;
	END_FOR
	TimerIntermittingLightOFF := TRUE;
	TimerIntermittingLightON := FALSE;
	TimerCabLightOFF := FALSE;
END_IF

IF(IntermittingLightOFF = TRUE AND StopOccurred = TRUE AND DesiredFloor = -1) THEN
	FOR i:= 0 TO N-1 DO
		Floor[i].CabLed := FALSE;
	END_FOR
	TimerIntermittingLightON := TRUE;
	TimerIntermittingLightOFF := FALSE;
	TimerCabLightOFF := FALSE;
END_IF

IF (DesiredFloor  <> -1 )  THEN
	TimerIntermittingLightON := FALSE;
	TimerIntermittingLightOFF := FALSE;
	TimerCabLightOFF := FALSE;
	Cabin.Light := TRUE;

	IF (StopOccurred = TRUE) THEN
		Stop_Management();
	ELSE
		Move_To(CurrentFloor, DesiredFloor);
	END_IF
END_IF
END_FUNCTION

(* POU Delete_All_Queue, ST *)
FUNCTION Delete_All_Queue: BOOL
VAR_INPUT
END_VAR
VAR
	i: INT;
END_VAR
FOR i:= 0 TO N-1 DO
	Queue[i] := -1;
	CabCall[i] := -1;
	UpCall[i] := -1;
	DwCall[i] := -1;
END_FOR
END_FUNCTION

(* POU Stop_Management, ST *)
FUNCTION Stop_Management: BOOL
VAR_INPUT
END_VAR
VAR
	i: INT;
END_VAR
FOR i:= 0 TO N-1 DO
	IF (Floor[i].CabPresence = TRUE) THEN
		Floor[i].CabLed := TRUE;
	ELSE
		Floor[i].CabLed := FALSE;
	END_IF
END_FOR

IF (CurrentFloor <> DesiredFloor ) THEN
	Move_To(CurrentFloor, DesiredFloor);
ELSIF (CurrentFloor = DesiredFloor) THEN
	IF (Floor[DesiredFloor].CabPresence = FALSE) THEN
		(*Elevator Between Floor 1 and 2*)
		FOR i:=0 TO N-2 DO
			IF (IsBetween[i] = TRUE AND DesiredFloor = i) THEN
				Cabin.GoDown := TRUE;
				MovingUp := FALSE;
				MovingDw := TRUE;
				MovedUp := FALSE;
				MovedDw := TRUE;
				Displacement := Displacement +1;
			ELSIF(IsBetween[i] = TRUE AND DesiredFloor = i+1) THEN
				Cabin.GoUp := TRUE;
				MovingUp := TRUE;
				MovingDw := FALSE;
				MovedUp := TRUE;
				MovedDw := FALSE;
				Displacement := Displacement -1;
			END_IF
		END_FOR
	ELSIF (Floor[DesiredFloor].CabPresence = TRUE) THEN
		Cabin.GoDown:= FALSE;
		Cabin.GoUp:= FALSE;
		MovingUp := FALSE;
		MovingDw := FALSE;
	END_IF
END_IF
END_FUNCTION

(* POU Move_To, ST *)
FUNCTION Move_To: BOOL
VAR_INPUT
	CurFloor: INT;
	DesFloor: INT;
END_VAR
VAR
	i: INT := 0;
	FloorDifference: INT;
END_VAR
FloorDifference := DesFloor  - CurFloor;

IF (FloorDifference > 0) THEN
	Cabin.GoUp := TRUE;
	MovingUp := TRUE;
	MovingDw := FALSE;
	MovedUp := TRUE;
	MovedDw := FALSE;
	Displacement := Displacement -1;
	FOR i := 0 TO (N-1) DO
		IF (Floor[i].CabPresence = TRUE)  THEN
			TimerErrorCabin := FALSE;
			EXIT;
		ELSE
			TimerErrorCabin := TRUE;
		END_IF
	END_FOR
ELSIF (FloorDifference < 0) THEN
	Cabin.GoDown := TRUE;
	MovingDw := TRUE;
	MovingUp := FALSE;
	MovedDw := TRUE;
	MovedUp := FALSE;
	Displacement := Displacement +1;
	FOR i := 0 TO (N-1) DO
		IF (Floor[i].CabPresence = TRUE)  THEN
			TimerErrorCabin := FALSE;
			EXIT;
		ELSE
			TimerErrorCabin := TRUE;
		END_IF
	END_FOR
ELSIF (FloorDifference = 0) THEN
	Cabin.GoDown := FALSE;
	Cabin.GoUp := FALSE;
	MovingUp := FALSE;
	MovingDw := FALSE;
	TimerErrorCabin := FALSE;
END_IF
END_FUNCTION

(* POU Doors_Management_No_Obstacle, ST *)
FUNCTION Doors_Management_No_Obstacle: BOOL
VAR_INPUT
END_VAR
VAR
	i: INT;
END_VAR
IF (DesiredFloor  = CurrentFloor  AND Cabin.GoDown = FALSE AND Cabin.GoUp = FALSE) THEN
	IF(EndOpening = FALSE) THEN
		EndOpening := Open_Door(CurrentFloor);
		StopOccurred := FALSE;
		EndMovement := FALSE;

		FOR i:=0 TO N-1 DO
			TimerErrorClosingDoor[i] := FALSE;
			IF(CurrentFloor = i) THEN
				TimerErrorOpeningDoor[i] := TRUE;
			ELSE
				TimerErrorOpeningDoor[i]:= FALSE;
			END_IF
		END_FOR
	END_IF

       IF (Cabin.GoUp = FALSE AND Cabin.GoDown = FALSE) THEN
		i:= 0;
		IF ((Cabin.Call[i] = TRUE OR Floor[i].CallUp = TRUE)  AND Floor[i].CabPresence = TRUE ) THEN
			EndMovement := FALSE;
			EndOpening := FALSE;
			Floor[i].DoorClose := FALSE;
			TimerDoor := FALSE;
			TimerErrorOpeningDoor[i] := TRUE;
			TimerErrorClosingDoor[i] := FALSE;
		END_IF

		FOR i:= 1 TO N-2 DO
	     		IF ((Cabin.Call[i] = TRUE OR Floor[i].CallUp = TRUE OR Floor[i].CallDw = TRUE) AND Floor[i].CabPresence = TRUE ) THEN
				EndMovement := FALSE;
				EndOpening := FALSE;
				Floor[i].DoorClose := FALSE;
				TimerDoor := FALSE;
				TimerErrorOpeningDoor[i] := TRUE;
				TimerErrorClosingDoor[i] := FALSE;
			END_IF
		END_FOR
		i:= N-1;
		IF ((Cabin.Call[i] = TRUE OR Floor[i].CallDw = TRUE) AND Floor[i].CabPresence = TRUE ) THEN
			EndMovement := FALSE;
			EndOpening := FALSE;
			Floor[i].DoorClose := FALSE;
			TimerDoor := FALSE;
			TimerErrorOpeningDoor[i] := TRUE;
			TimerErrorClosingDoor[i] := FALSE;
		END_IF
	END_IF
END_IF

IF(EndOpening = TRUE) THEN
	FOR i:= 0 TO N-1 DO
		TimerErrorOpeningDoor[i] := FALSE;
	END_FOR
END_IF

IF (DesiredFloor = CurrentFloor  AND StartClose = TRUE) THEN
	FOR i:= 0 TO N-1 DO
		IF(CurrentFloor = i) THEN
			TimerErrorClosingDoor[i] := TRUE;
		END_IF
	END_FOR
	EndMovement := Close_Door(CurrentFloor);
END_IF

IF (EndMovement = TRUE AND DesiredFloor = CurrentFloor AND ReadyToDelete = FALSE) THEN
	i:= 0;
	IF ((Cabin.Call[i] = TRUE OR Floor[i].CallUp = TRUE) AND CurrentFloor = i) THEN
		EndMovement := FALSE;
		EndOpening := FALSE;
		Floor[i].DoorClose := FALSE;
		TimerDoor := FALSE;
		TimerErrorOpeningDoor[i] := TRUE;
		TimerErrorClosingDoor[i] := FALSE;
	END_IF
	FOR i:= 1 TO N-2 DO
		IF ((Cabin.Call[i] = TRUE OR Floor[i].CallUp = TRUE OR Floor[i].CallDw = TRUE) AND CurrentFloor = i) THEN
			EndMovement := FALSE;
			EndOpening := FALSE;
			Floor[i].DoorClose := FALSE;
			TimerDoor := FALSE;
			TimerErrorOpeningDoor[i] := TRUE;
			TimerErrorClosingDoor[i] := FALSE;
		END_IF
	END_FOR

	i := N-1 ;
	IF ((Cabin.Call[i] = TRUE OR Floor[i].CallDw = TRUE) AND CurrentFloor = i) THEN
		EndMovement := FALSE;
		EndOpening := FALSE;
		Floor[i].DoorClose := FALSE;
		TimerDoor := FALSE;
		TimerErrorOpeningDoor[i] := TRUE;
		TimerErrorClosingDoor[i] := FALSE;
	END_IF
END_IF

IF (EndMovement = TRUE AND DesiredFloor = CurrentFloor AND ReadyToDelete = TRUE) THEN
	DesiredFloor := -1;
	EndMovement := FALSE;
	EndOpening := FALSE;
	FOR i:= 0 TO N-1 DO
		TimerErrorClosingDoor[i] := FALSE;
	END_FOR
	TimerCabLightOFF := TRUE;
	Floor[CurrentFloor].LedDw := FALSE;
	Floor[CurrentFloor].LedUp := FALSE;
	IF (Multiple = TRUE) THEN
		Delete_To_Queue();
	END_IF
	IF (Optimized = TRUE) THEN
		Delete_To_Calls();
	END_IF
END_IF
END_FUNCTION

(* POU Open_Door, ST *)
FUNCTION Open_Door: BOOL
VAR_INPUT
	CurFloor: UINT;
END_VAR
VAR
END_VAR
IF (Floor[CurFloor].DoorOpened = FALSE) THEN
	Floor[CurFloor].DoorOpen := TRUE;
	IF (Displacement = 450) THEN
		Door0 := Door0 + 1;
	ELSIF (Displacement = 300) THEN
		Door1 := Door1 + 1;
	ELSIF (Displacement = 150) THEN
		Door2 := Door2 + 1;
	ELSIF (Displacement = 0) THEN
		Door3 := Door3 + 1;
	END_IF
ELSE
	Floor[CurFloor].DoorOpen := FALSE;
END_IF

IF (Floor[CurFloor].DoorOpened = TRUE) THEN
	TimerDoor := TRUE;
	Open_Door := TRUE;
ELSE
	Open_Door := FALSE;
END_IF
END_FUNCTION

(* POU Close_Door, ST *)
FUNCTION Close_Door: BOOL
VAR_INPUT
	CurFloor: UINT;
END_VAR
VAR
END_VAR
IF (Floor[CurFloor].DoorClosed = FALSE  AND Cabin.Obstacle = FALSE) THEN
	Floor[CurFloor].DoorClose := TRUE;
	IF (Displacement = 450) THEN
		Door0 := Door0 - 1;
	ELSIF (Displacement = 300) THEN
		Door1 := Door1 - 1;
	ELSIF (Displacement = 150) THEN
		Door2 := Door2 - 1;
	ELSIF (Displacement = 0) THEN
		Door3 := Door3 - 1;
	END_IF
ELSE
	Floor[CurFloor].DoorClose := FALSE;
END_IF

IF (Floor[CurFloor].DoorClosed = TRUE) THEN
	TimerDoor := FALSE;
	Close_Door := TRUE;
ELSE
	Close_Door := FALSE;
END_IF
END_FUNCTION

(* POU Delete_To_Queue, ST *)
FUNCTION Delete_To_Queue: BOOL
VAR_INPUT
END_VAR
VAR
	i: INT;
	j: INT := 0;
	TemporaryArray: ARRAY [0..5] OF INT; (*==============================================================*)
	SwapDone: BOOL := FALSE;
END_VAR
IF (CurrentFloor = 0) THEN
	Floor[CurrentFloor].LedUp := FALSE;
ELSIF (CurrentFloor = N-1) THEN
	Floor[CurrentFloor].LedDw := FALSE;
ELSE
	Floor[CurrentFloor].LedDw := FALSE;
	Floor[CurrentFloor].LedUp := FALSE;
END_IF

FOR i := 0 TO N-1  DO
	IF (Queue[i] = CurrentFloor) THEN
		Queue[i] := -2;
	END_IF
END_FOR

FOR i := 0 TO N-1 DO
	SwapDone := FALSE;
	IF (j <= N-1) THEN
		WHILE (swapDone = FALSE) DO
			IF (Queue[j] <> -2 ) THEN
				TemporaryArray[i] := Queue[j];
				SwapDone := TRUE;
				j := j+1;
			ELSE
				j := j+1;
			END_IF
		END_WHILE
	ELSE
		TemporaryArray[i] := -1;
	END_IF
END_FOR

Queue:= temporaryArray;
Delete_To_Queue := TRUE;
END_FUNCTION

(* POU Delete_To_Calls, ST *)
FUNCTION Delete_To_Calls: BOOL
VAR_INPUT
END_VAR
VAR
	i: INT;
	j: INT := 0;
	k: INT := 0;
	l: INT := 0;
	TemporaryArray1: ARRAY [0..5] OF INT;(*==============================================================*)
	TemporaryArray2: ARRAY [0..5] OF INT;(*==============================================================*)
	TemporaryArray3: ARRAY [0..5] OF INT;(*==============================================================*)
	SwapDone1: BOOL := FALSE;
	SwapDone2: BOOL := FALSE;
	SwapDone3: BOOL := FALSE;
END_VAR
IF (CurrentFloor = 0) THEN
	Floor[CurrentFloor].LedUp := FALSE;
ELSIF (CurrentFloor = N-1) THEN
	Floor[CurrentFloor].LedDw := FALSE;
ELSE
	Floor[CurrentFloor].LedUp := FALSE;
	Floor[CurrentFloor].LedDw := FALSE;
END_IF

FOR i := 0 TO N-1 DO
	IF (CabCall[i] = CurrentFloor) THEN
		CabCall[i] := -2;
	END_IF
	IF (UpCall[i] = CurrentFloor) THEN
		UpCall[i] := -2;
	END_IF
	IF (DwCall[i] = CurrentFloor) THEN
		DwCall[i] := -2;
	END_IF
END_FOR

FOR i := 0 TO N-1 DO
	SwapDone1 := FALSE;
	SwapDone2 := FALSE;
	SwapDone3 := FALSE;

	IF (j <= N-1) THEN
		WHILE (SwapDone1 = FALSE) DO
			IF (CabCall[j] <> -2) THEN
				TemporaryArray1[i] := CabCall[j];
				SwapDone1 := TRUE;
			END_IF
			j := j+1;
		END_WHILE
	ELSE
		TemporaryArray1[i] := -1;
	END_IF

	IF (k <= N-1) THEN
		WHILE (SwapDone2 = FALSE) DO
			IF (UpCall[k] <> -2) THEN
				TemporaryArray2[i] := UpCall[k];
				SwapDone2 := TRUE;
			END_IF
			k := k+1;
		END_WHILE
	ELSE
		TemporaryArray2[i] := -1;
	END_IF

	IF (l <= N-1) THEN
		WHILE (SwapDone3 = FALSE) DO
			IF (DwCall[l] <> -2) THEN
				TemporaryArray3[i] := DwCall[l];
				SwapDone3 := TRUE;
			END_IF
			l := l+1;
		END_WHILE
	ELSE
		TemporaryArray3[i] := -1;
	END_IF
END_FOR

CabCall := TemporaryArray1;
UpCall := TemporaryArray2;
DwCall := TemporaryArray3;

Delete_To_Calls := TRUE;
END_FUNCTION

(* POU Obstacle_Function, ST *)
FUNCTION Obstacle_Function: BOOL
VAR_INPUT
END_VAR
VAR
END_VAR
IF (Floor[CurrentFloor].DoorClose = TRUE AND Cabin.Obstacle = TRUE) THEN
	TimerDoorAfterObstacle := FALSE;
END_IF

IF (Cabin.Obstacle = TRUE) THEN
	TimerDoorAfterObstacle := FALSE;
	ObstacleOccurred := TRUE;
	ObstacleCase := TRUE;
	Floor[CurrentFloor].DoorClose := FALSE;
END_IF
END_FUNCTION

(* POU Doors_Management_Obstacle, ST *)
FUNCTION Doors_Management_Obstacle: BOOL
VAR_INPUT
END_VAR
VAR
	i: INT;
END_VAR
IF ((Cabin.Obstacle = TRUE OR ObstacleOccurred = TRUE) AND EndOpeningObstacle = FALSE) THEN
	EndOpeningObstacle := Open_Door(CurrentFloor);
	StopOccurred := FALSE;
	EndMovement := FALSE;

	FOR i := 0 TO N-1 DO
		TimerErrorClosingDoor[i] := FALSE;
		IF(CurrentFloor = i) THEN
			TimerErrorOpeningDoor[i] := TRUE;
		ELSE
			TimerErrorOpeningDoor[i] := FALSE;
		END_IF
	END_FOR
	Cabin.Light := TRUE;
END_IF

IF (EndOpeningObstacle = TRUE) THEN
	FOR i := 0 TO N-1 DO
		TimerErrorOpeningDoor[i]:= FALSE;
	END_FOR
END_IF

IF (Cabin.Obstacle = FALSE) THEN
	IF(Cabin.GoUp = FALSE AND Cabin.GoDown = FALSE) THEN
		i:= 0;
		IF ((Cabin.Call[i] = TRUE OR Floor[i].CallUp = TRUE)  AND Floor[i].CabPresence = TRUE  ) THEN
			TimerDoorAfterObstacle := FALSE;
			EndOpeningObstacle := FALSE;
			ObstacleOccurred := TRUE;
			Floor[i].DoorClose := FALSE;
			TimerDoor := FALSE;
			TimerErrorOpeningDoor[i] := TRUE;
			TimerErrorClosingDoor[i] := FALSE;
		END_IF
		FOR i:= 1 TO N-2 DO
			IF ((Cabin.Call[i] = TRUE OR Floor[i].CallUp = TRUE OR Floor[i].CallDw = TRUE) AND Floor[i].CabPresence = TRUE ) THEN
				TimerDoorAfterObstacle := FALSE;
				EndOpeningObstacle := FALSE;
				ObstacleOccurred := TRUE;
				Floor[1].DoorClose := FALSE;
				TimerDoor := FALSE;
				TimerErrorOpeningDoor[i] := TRUE;
				TimerErrorClosingDoor[i] := FALSE;
			END_IF
		END_FOR
		i:= N-1;
		IF ((Cabin.Call[i] = TRUE OR Floor[i].CallDw = TRUE) AND Floor[i].CabPresence = TRUE ) THEN
			TimerDoorAfterObstacle := FALSE;
			EndOpeningObstacle := FALSE;
			ObstacleOccurred := TRUE;
			Floor[i].DoorClose := FALSE;
			TimerDoor := FALSE;
			TimerErrorOpeningDoor[i] := TRUE;
			TimerErrorClosingDoor[i] := FALSE;
		END_IF
	END_IF


	 IF (EndOpeningObstacle = TRUE) THEN
		TimerDoorAfterObstacle := TRUE;
		EndOpeningObstacle := FALSE;
		ObstacleOccurred := FALSE;
	END_IF

	IF (StartCloseAfterObstacle = TRUE) THEN
		EndMovementObstacle := Close_Door(CurrentFloor);
		FOR i:= 0 TO N-1 DO
			IF(CurrentFloor = i) THEN
				TimerErrorClosingDoor[i] := TRUE;
			END_IF
		END_FOR
	END_IF

	IF (EndMovementObstacle = TRUE AND DesiredFloor = CurrentFloor AND ReadyToDelete = FALSE) THEN
		i:= 0;
		IF ((Cabin.Call[i] = TRUE OR Floor[i].CallUp = TRUE) AND CurrentFloor = i) THEN
			EndMovementObstacle := FALSE;
			EndOpeningObstacle := FALSE;
			Floor[i].DoorClose := FALSE;
			TimerDoor := FALSE;
			TimerDoorAfterObstacle := FALSE;
			TimerErrorOpeningDoor[i] := TRUE;
			TimerErrorClosingDoor[i] := FALSE;
		END_IF
		FOR i:= 1 TO N-2 DO
			IF ((Cabin.Call[i] = TRUE OR Floor[i].CallUp = TRUE OR Floor[i].CallDw = TRUE) AND CurrentFloor = i) THEN
				EndMovementObstacle := FALSE;
				EndOpeningObstacle := FALSE;
				Floor[i].DoorClose := FALSE;
				TimerDoor := FALSE;
				TimerDoorAfterObstacle := FALSE;
				TimerErrorOpeningDoor[i] := TRUE;
				TimerErrorClosingDoor[i] := FALSE;
			END_IF
		END_FOR
		i:= N-1;
		IF ((Cabin.Call[i] = TRUE OR Floor[i].CallDw = TRUE) AND CurrentFloor = i) THEN
			EndMovementObstacle := FALSE;
			EndOpeningObstacle := FALSE;
			Floor[i].DoorClose := FALSE;
			TimerDoor := FALSE;
			TimerDoorAfterObstacle := FALSE;
			TimerErrorOpeningDoor[i] := TRUE;
			TimerErrorClosingDoor[i] := FALSE;
		END_IF
	END_IF

	IF (EndMovementObstacle = TRUE AND DesiredFloor = CurrentFloor AND ReadyToDelete = TRUE) THEN
		TimerDoorAfterObstacle := FALSE;
		ObstacleCase := FALSE;
		EndMovementObstacle := FALSE;
		DesiredFloor := -1;
		EndMovement := FALSE;
		EndOpening := FALSE;
		FOR i:= 0 TO N-1 DO
			TimerErrorClosingDoor[i] := FALSE;
		END_FOR
		TimerCabLightOFF := TRUE;
		Floor[CurrentFloor].LedDw := FALSE;
		Floor[CurrentFloor].LedUp := FALSE;
		IF (Multiple = TRUE) THEN
			Delete_To_Queue();
		END_IF
		IF (Optimized = TRUE) THEN
			Delete_To_Calls();
		END_IF
	END_IF
END_IF
END_FUNCTION

(* POU Error_Management, ST *)
FUNCTION Error_Management: BOOL
VAR_INPUT
END_VAR
VAR
	i: INT;
END_VAR
Cabin.GoDown := FALSE;
Cabin.GoUp := FALSE;

FOR i := 0 TO N-1 DO
	Floor[i].DoorOpen := FALSE;
	Floor[i].DoorClose := FALSE;
END_FOR

IF (TimerIntermittingLightOFF = FALSE) THEN
	TimerIntermittingLightON := TRUE;
END_IF

IF(IntermittingLightON = TRUE) THEN
	FOR i:= 0 TO N-1 DO
		Floor[i].CabLed := TRUE;
	END_FOR
	TimerIntermittingLightOFF := TRUE;
	TimerIntermittingLightON := FALSE;
END_IF

IF(IntermittingLightOFF = TRUE) THEN
	FOR i:= 0 TO N-1 DO
		Floor[i].CabLed := FALSE;
	END_FOR
	TimerIntermittingLightON := TRUE;
	TimerIntermittingLightOFF := FALSE;
END_IF
END_FUNCTION

(* POU ASS_OUTPUT, ST *)
PROGRAM ASS_OUTPUT
VAR
END_VAR
(*Floor 0 Assignment*)
Floor0DoorOpen			:= Floor[0].DoorOpen;
Floor0DoorClose			:= Floor[0].DoorClose;
CabLed0 					:= Floor[0].CabLed;
Floor0LedUp				:= Floor[0].LedUp;

(*Floor 1 Assignment*)
Floor1DoorOpen			:= Floor[1].DoorOpen;
Floor1DoorClose			:= Floor[1].DoorClose;
CabLed1 					:= Floor[1].CabLed;
Floor1LedDw				:= Floor[1].LedDw;
Floor1LedUp				:= Floor[1].LedUp;

(*Floor 2 Assignment*)
Floor2DoorOpen			:= Floor[2].DoorOpen;
Floor2DoorClose			:= Floor[2].DoorClose;
CabLed2 					:= Floor[2].CabLed;
Floor2LedDw				:= Floor[2].LedDw;
Floor2LedUp				:= Floor[2].LedUp;

(*Floor 3 Assignment*)
Floor3DoorOpen			:= Floor[3].DoorOpen;
Floor3DoorClose			:= Floor[3].DoorClose;
CabLed3 					:= Floor[3].CabLed;
Floor3LedDw				:= Floor[3].LedDw;

(*Cabin  Assignment*)
CabLight					:= Cabin.Light;
CabGoDown				:= Cabin.GoDown;
CabGoUp					:= Cabin.GoUp;
END_PROGRAM

(* POU HMI, ST *)
PROGRAM HMI
VAR
	i: BOOL;
END_VAR
(* Assignement variables of the inputs for the HMI *)

DoorClosed0 := Floor[0].DoorClosed;
DoorOpened0 := Floor[0].DoorOpened;
DoorClosed1 := Floor[1].DoorClosed;
DoorOpened1 := Floor[1].DoorOpened;
DoorClosed2 := Floor[2].DoorClosed;
DoorOpened2 := Floor[2].DoorOpened;
DoorClosed3 := Floor[3].DoorClosed;
DoorOpened3 := Floor[3].DoorOpened;

(* Assignement tag for the error *)

IF (ErrorClosingDoor[0] = TRUE) THEN
	Error := 1;
ELSIF (ErrorClosingDoor[1] = TRUE) THEN
	Error := 2;
ELSIF (ErrorClosingDoor[2] = TRUE) THEN
	Error := 3;
ELSIF (ErrorClosingDoor[3] = TRUE) THEN
	Error := 4;
ELSIF (ErrorOpeningDoor[0] = TRUE) THEN
	Error := 5;
ELSIF (ErrorOpeningDoor[1] = TRUE) THEN
	Error := 6;
ELSIF (ErrorOpeningDoor[2] = TRUE) THEN
	Error := 7;
ELSIF (ErrorOpeningDoor[3] = TRUE) THEN
	Error := 8;
ELSIF (Cabin.ErrorCabin = TRUE) THEN
	Error := 9;
ELSIF (Weight>LimitWeight = TRUE) THEN
	Error := 10;
ELSE
	Error := 0;
END_IF

(* Assignement order  for the calls *)
       IntCall1:= CabCall[0];
	IntCall2:= CabCall[1];
	IntCall3:= CabCall[2];
	IntCall4:= CabCall[3];
	UpCall1:=UpCall[0];
	UpCall2:=UpCall[1];
	UpCall3:=UpCall[2];
	UpCall4:=UpCall[3];
	DwCall1:=DwCall[0];
	DwCall2:=DwCall[1];
	DwCall3:=DwCall[2];
	DwCall4:=DwCall[3];
	Queue1:=Queue[0];
	Queue2:=Queue[1];
	Queue3:=Queue[2];
	Queue4:=Queue[3];

(* Defining tag for the position of the elevator *)


IF (currentFloor=0 AND isbetween[0]=FALSE) THEN
	floorIndicator:=0;
END_IF

IF ( isbetween[0]=TRUE) THEN
	floorIndicator:=1;
END_IF

IF (currentFloor=1 AND isbetween[0]=FALSE AND isbetween[1]=FALSE) THEN
	floorIndicator:=2;
END_IF

IF ( isbetween[1]=TRUE) THEN
	floorIndicator:=3;
END_IF

IF (currentFloor=2 AND isbetween[1]=FALSE AND isbetween[2]=FALSE) THEN
	floorIndicator:=4;
END_IF

IF ( isbetween[2]=TRUE) THEN
	floorIndicator:=5;
END_IF

IF (currentFloor=3 AND isbetween[2]=FALSE) THEN
	floorIndicator:=6;
END_IF
END_PROGRAM

(* POU MANUAL, ST *)
PROGRAM MANUAL
VAR
END_VAR
Define_Current_Floor(StopOccurred);

IF (GoUp = TRUE) THEN
	Cabin.GoUp := TRUE;
ELSE
	Cabin.GoUp := FALSE;
END_IF

IF (GoDw = TRUE) THEN
	Cabin.GoDown := TRUE;
ELSE
	Cabin.GoDown := FALSE;
END_IF

IF (Open0 = TRUE) THEN
	Floor[0].DoorOpen := TRUE;
ELSE
	Floor[0].DoorOpen := FALSE;
END_IF

IF (Open1 = TRUE) THEN
	Floor[1].DoorOpen := TRUE;
ELSE
	Floor[1].DoorOpen := FALSE;
END_IF

IF (Open2 = TRUE) THEN
	Floor[2].DoorOpen := TRUE;
ELSE
	Floor[2].DoorOpen := FALSE;
END_IF

IF (Open3 = TRUE) THEN
	Floor[3].DoorOpen := TRUE;
ELSE
	Floor[3].DoorOpen := FALSE;
END_IF

IF (Close0 = TRUE) THEN
	Floor[0].DoorClose := TRUE;
ELSE
	Floor[0].DoorClose := FALSE;
END_IF

IF (Close1 = TRUE) THEN
	Floor[1].DoorClose := TRUE;
ELSE
	Floor[1].DoorClose := FALSE;
END_IF

IF (Close2 = TRUE) THEN
	Floor[2].DoorClose := TRUE;
ELSE
	Floor[2].DoorClose := FALSE;
END_IF

IF (Close3 = TRUE) THEN
	Floor[3].DoorClose := TRUE;
ELSE
	Floor[3].DoorClose := FALSE;
END_IF
END_PROGRAM

(* Visualisation Dynamic_Simulation
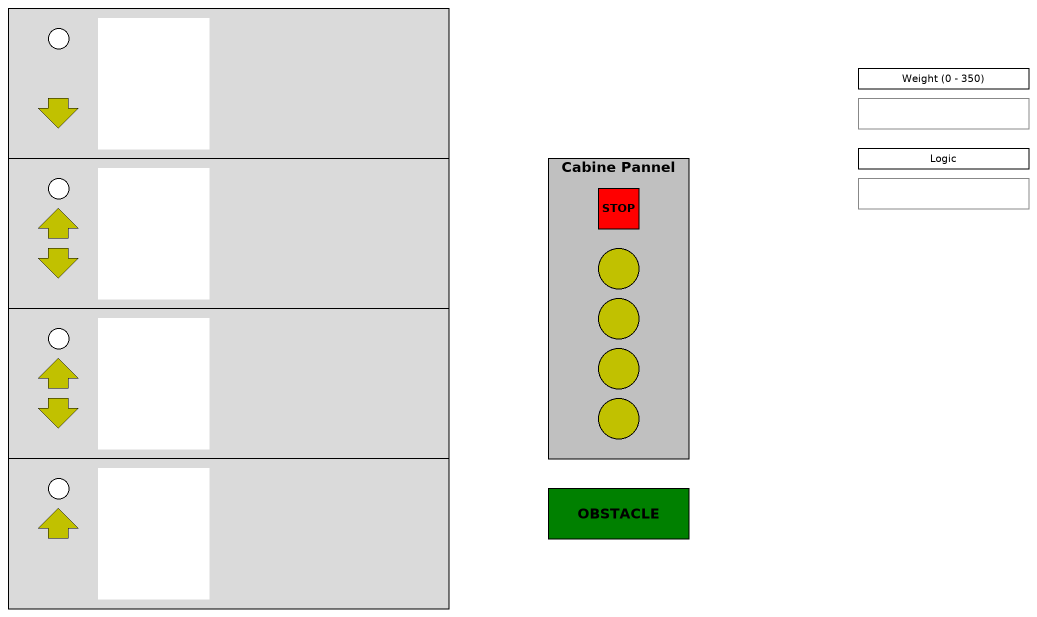
ellipse at (100,330)-(121,351): alarm colour if .CabLed1
ellipse at (100,480)-(121,501): alarm colour if .CabLed0
ellipse at (100,180)-(121,201): alarm colour if .CabLed2
ellipse at (100,30)-(121,51): alarm colour if .CabLed3
rectangle at (600,160)-(741,461): text "Cabine Pannel"
rectangle at (650,190)-(691,231): text "STOP"; taps .CabStop
rounded rectangle at (600,490)-(741,541): text "OBSTACLE"; alarm colour if .CabObstacle; toggles .CabObstacle
rectangle at (150,20)-(261,151): alarm colour if .CabLight; y offset .Displacement
rectangle at (150,20)-(261,151): x offset .Door3
rectangle at (150,170)-(261,301): x offset .Door2
rectangle at (150,320)-(261,451): x offset .Door1
rectangle at (150,470)-(261,601): x offset .Door0
polygon at (90,400)-(130,430): alarm colour if .Floor1LedDw; taps .Floor1DwBt
polygon at (90,250)-(130,280): alarm colour if .Floor2LedDw; taps .Floor2DwBt
polygon at (90,100)-(130,130): alarm colour if .Floor3LedDw; taps .Floor3DwBt
polygon at (90,210)-(130,240): alarm colour if .Floor2LedUp; taps .Floor2UpBt
polygon at (90,360)-(130,390): alarm colour if .Floor1LedUp; taps .Floor1UpBt
polygon at (90,510)-(130,540): alarm colour if .Floor0LedUp; taps .Floor0UpBt
ellipse at (650,250)-(691,291): alarm colour if .CabLed3; taps .CabCallP3
ellipse at (650,300)-(691,341): alarm colour if .CabLed2; taps .CabCallP2
ellipse at (650,350)-(691,391): alarm colour if .CabLed1; taps .CabCallP1
ellipse at (650,400)-(691,441): alarm colour if .CabLed0; taps .CabCallP0
rectangle at (910,150)-(1081,171): text "Logic"
rectangle at (910,70)-(1081,91): text "Weight (0 - 350)"
6 more shapes without text or variables
5 elements of other kinds (tables, trends, ...) not read
*)

(* Visualisation Static_Simulation
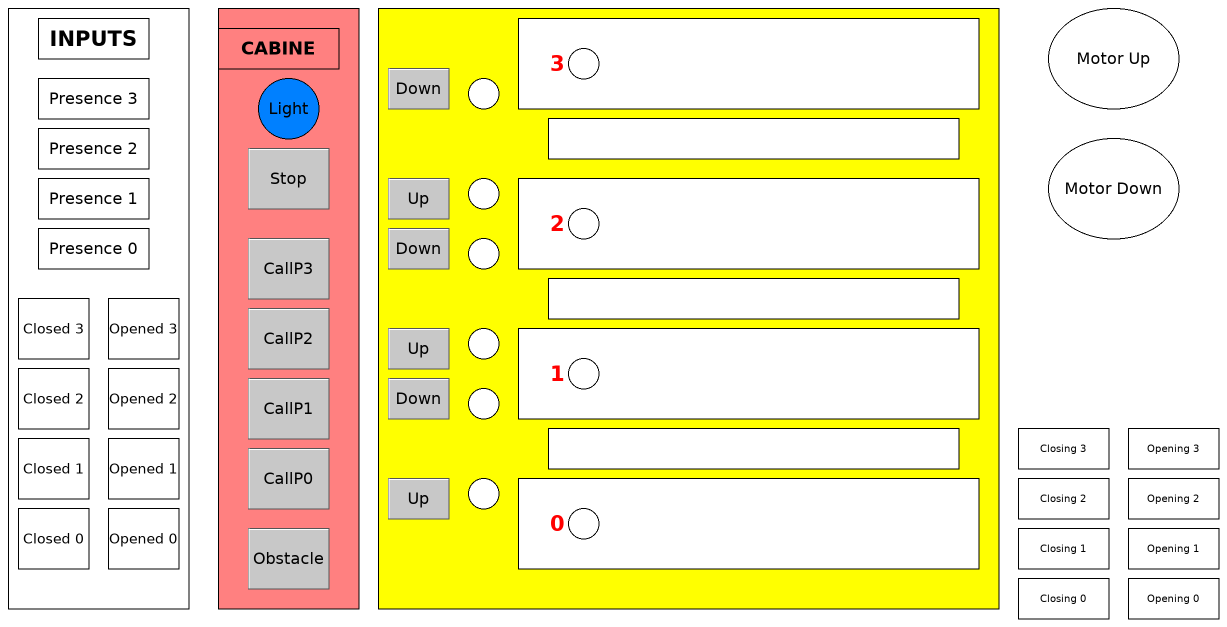
button at (260,250)-(341,311): text "CallP3"; taps .CabCallP3
button at (260,320)-(341,381): text "CallP2"; taps .CabCallP2
button at (260,390)-(341,451): text "CallP1"; taps .CabCallP1
button at (260,460)-(341,521): text "CallP0"; taps .CabCallP0
button at (260,540)-(341,601): text "Obstacle"; toggles .CabObstacle
button at (260,160)-(341,221): text "Stop"; taps .CabStop
ellipse at (270,90)-(331,151): text "Light"; alarm colour if .CabLight
rectangle at (230,40)-(351,81): text "CABINE"
rectangle at (530,30)-(991,121): text "3"; alarm colour if .Floor3CabPresence
rectangle at (530,190)-(991,281): text "2"; alarm colour if .Floor2CabPresence
rectangle at (530,340)-(991,431): text "1"; alarm colour if .Floor1CabPresence
rectangle at (530,490)-(991,581): text "0"; alarm colour if .Floor0CabPresence
rectangle at (560,130)-(971,171): alarm colour if .isBetween[2]
rectangle at (560,290)-(971,331): alarm colour if .isBetween[1]
rectangle at (560,440)-(971,481): alarm colour if .isBetween[0]
rectangle at (710,40)-(781,111): alarm colour if .Floor3DoorClosed
rectangle at (710,200)-(781,271): alarm colour if .Floor2DoorClosed
rectangle at (710,350)-(781,421): alarm colour if .Floor1DoorClosed
rectangle at (710,500)-(781,571): alarm colour if .Floor0DoorClosed
rectangle at (840,40)-(911,111): alarm colour if .Floor3DoorOpened
rectangle at (840,200)-(911,271): alarm colour if .Floor2DoorOpened
rectangle at (840,350)-(911,421): alarm colour if .Floor1DoorOpened
rectangle at (840,500)-(911,571): alarm colour if .Floor0DoorOpened
ellipse at (580,60)-(611,91): alarm colour if .CabLed3
ellipse at (580,220)-(611,251): alarm colour if .CabLed2
ellipse at (580,370)-(611,401): alarm colour if .CabLed1
ellipse at (580,520)-(611,551): alarm colour if .CabLed0
button at (400,80)-(461,121): text "Down"; taps Floor3DwBt
button at (400,240)-(461,281): text "Down"; taps Floor2DwBt
button at (400,390)-(461,431): text "Down"; taps Floor1DwBt
button at (400,190)-(461,231): text "Up"; taps Floor2UpBt
button at (400,340)-(461,381): text "Up"; taps Floor1UpBt
button at (400,490)-(461,531): text "Up"; taps Floor0UpBt
ellipse at (480,90)-(511,121): alarm colour if Floor2LedDw
ellipse at (480,490)-(511,521): alarm colour if Floor0LedUp
ellipse at (480,340)-(511,371): alarm colour if Floor1LedUp
ellipse at (480,190)-(511,221): alarm colour if Floor2LedUp
ellipse at (480,400)-(511,431): alarm colour if Floor1LedDw
ellipse at (480,250)-(511,281): alarm colour if Floor2LedDw
ellipse at (1060,20)-(1191,121): text "Motor Up"; alarm colour if .CabGoUp
ellipse at (1060,150)-(1191,251): text "Motor Down"; alarm colour if .CabGoDown
rectangle at (50,90)-(161,131): text "Presence 3"; toggles .Floor3CabPresence
rectangle at (50,190)-(161,231): text "Presence 1"; toggles .Floor1CabPresence
rectangle at (50,140)-(161,181): text "Presence 2"; toggles .Floor2CabPresence
rectangle at (50,240)-(161,281): text "Presence 0"; toggles .Floor0CabPresence
rectangle at (120,310)-(191,371): text "Opened 3"; toggles .Floor3DoorOpened
rectangle at (120,380)-(191,441): text "Opened 2"; toggles .Floor2DoorOpened
rectangle at (120,450)-(191,511): text "Opened 1"; toggles .Floor1DoorOpened
rectangle at (120,520)-(191,581): text "Opened 0"; toggles .Floor0DoorOpened
rectangle at (30,310)-(101,371): text "Closed 3"; toggles .Floor3DoorClosed
rectangle at (30,380)-(101,441): text "Closed 2"; toggles .Floor2DoorClosed
rectangle at (30,450)-(101,511): text "Closed 1"; toggles .Floor1DoorClosed
rectangle at (30,520)-(101,581): text "Closed 0"; toggles .Floor0DoorClosed
rectangle at (50,30)-(161,71): text "INPUTS"
rounded rectangle at (1030,440)-(1121,481): text "Closing 3"; alarm colour if .Floor3DoorClose
rounded rectangle at (1030,490)-(1121,531): text "Closing 2"; alarm colour if .Floor2DoorClose
rounded rectangle at (1030,590)-(1121,631): text "Closing 0"; alarm colour if .Floor0DoorClose
rounded rectangle at (1030,540)-(1121,581): text "Closing 1"; alarm colour if .Floor1DoorClose
rounded rectangle at (1140,440)-(1231,481): text "Opening 3"; alarm colour if .Floor3DoorOpen
rounded rectangle at (1140,490)-(1231,531): text "Opening 2"; alarm colour if .Floor2DoorOpen
rounded rectangle at (1140,590)-(1231,631): text "Opening 0"; alarm colour if .Floor0DoorOpen
rounded rectangle at (1140,540)-(1231,581): text "Opening 1"; alarm colour if .Floor1DoorOpen
3 more shapes without text or variables
6 elements of other kinds (tables, trends, ...) not read
*)

(* Visualisation Static_Simulation_5_Floor
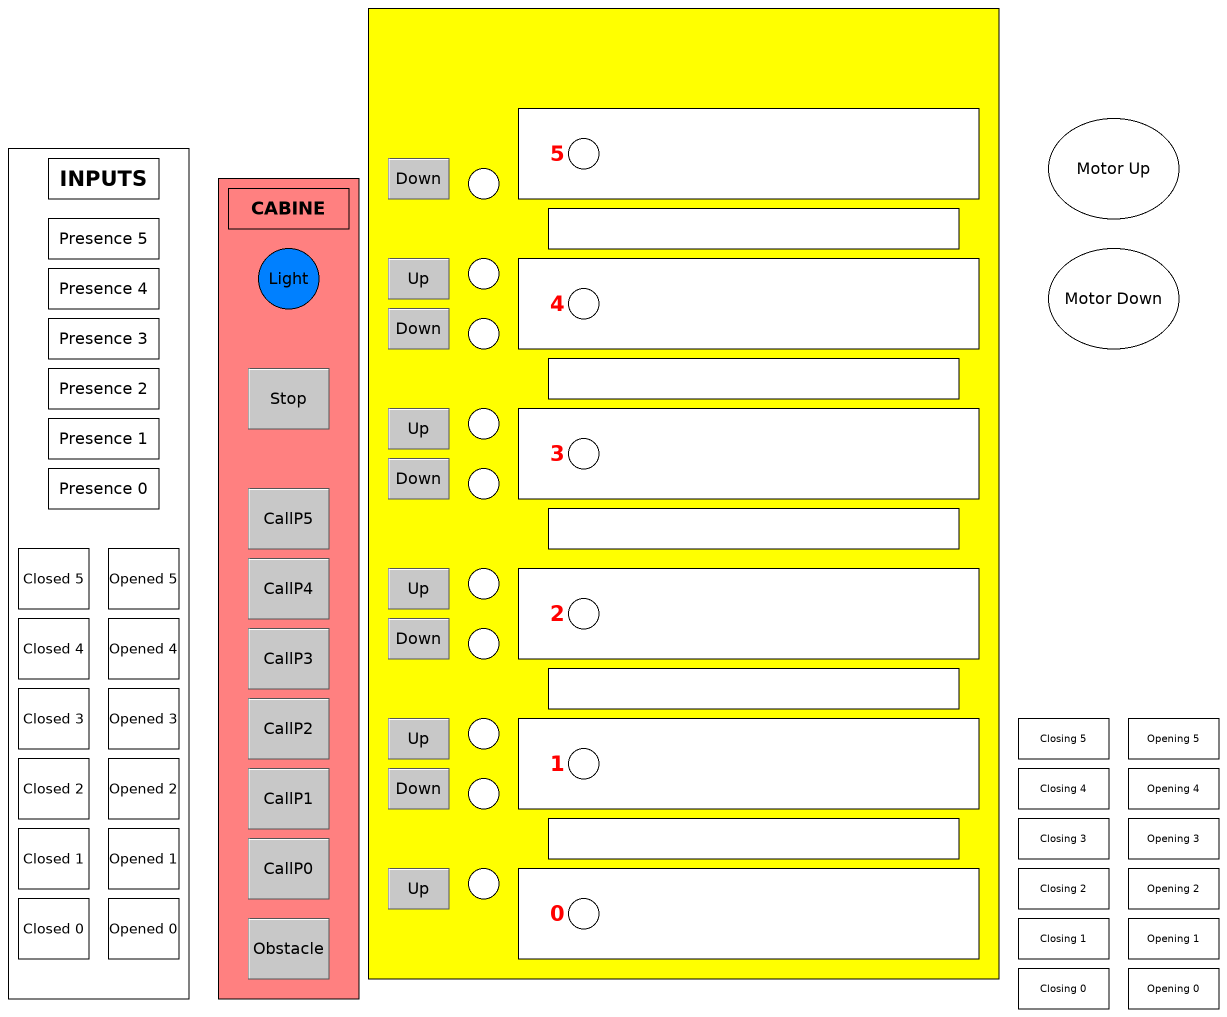
button at (290,630)-(371,691): text "CallP3"; taps .CabCallP3
button at (290,700)-(371,761): text "CallP2"; taps .CabCallP2
button at (290,770)-(371,831): text "CallP1"; taps .CabCallP1
button at (290,840)-(371,901): text "CallP0"; taps .CabCallP0
button at (290,920)-(371,981): text "Obstacle"; toggles .CabObstacle
button at (290,370)-(371,431): text "Stop"; taps .CabStop
ellipse at (300,250)-(361,311): text "Light"; alarm colour if .CabLight
rectangle at (270,190)-(391,231): text "CABINE"
rectangle at (560,410)-(1021,501): text "3"; alarm colour if .Floor[3].CabPresence
rectangle at (560,570)-(1021,661): text "2"; alarm colour if .Floor2CabPresence
rectangle at (560,720)-(1021,811): text "1"; alarm colour if .Floor1CabPresence
rectangle at (560,870)-(1021,961): text "0"; alarm colour if .Floor0CabPresence
rectangle at (590,510)-(1001,551): alarm colour if .isBetween[2]
rectangle at (590,670)-(1001,711): alarm colour if .isBetween[1]
rectangle at (590,820)-(1001,861): alarm colour if .isBetween[0]
rectangle at (740,420)-(811,491): alarm colour if Floor[3].DoorClosed
rectangle at (740,580)-(811,651): alarm colour if .Floor2DoorClosed
rectangle at (740,730)-(811,801): alarm colour if .Floor1DoorClosed
rectangle at (740,880)-(811,951): alarm colour if .Floor0DoorClosed
rectangle at (870,420)-(941,491): alarm colour if .Floor3DoorOpened
rectangle at (870,580)-(941,651): alarm colour if .Floor2DoorOpened
rectangle at (870,730)-(941,801): alarm colour if .Floor1DoorOpened
rectangle at (870,880)-(941,951): alarm colour if .Floor0DoorOpened
ellipse at (610,440)-(641,471): alarm colour if .CabLed3
ellipse at (610,600)-(641,631): alarm colour if .CabLed2
ellipse at (610,750)-(641,781): alarm colour if .CabLed1
ellipse at (610,900)-(641,931): alarm colour if .CabLed0
button at (430,460)-(491,501): text "Down"; taps Floor3DwBt
button at (430,620)-(491,661): text "Down"; taps Floor2DwBt
button at (430,770)-(491,811): text "Down"; taps Floor1DwBt
button at (430,570)-(491,611): text "Up"; taps Floor2UpBt
button at (430,720)-(491,761): text "Up"; taps Floor1UpBt
button at (430,870)-(491,911): text "Up"; taps Floor0UpBt
ellipse at (510,470)-(541,501): alarm colour if Floor2LedDw
ellipse at (510,870)-(541,901): alarm colour if Floor0LedUp
ellipse at (510,720)-(541,751): alarm colour if Floor1LedUp
ellipse at (510,570)-(541,601): alarm colour if Floor2LedUp
ellipse at (510,780)-(541,811): alarm colour if Floor1LedDw
ellipse at (510,630)-(541,661): alarm colour if Floor2LedDw
ellipse at (1090,120)-(1221,221): text "Motor Up"; alarm colour if .CabGoUp
ellipse at (1090,250)-(1221,351): text "Motor Down"; alarm colour if .CabGoDown
rectangle at (90,320)-(201,361): text "Presence 3"; toggles .Floor3CabPresence
rectangle at (90,420)-(201,461): text "Presence 1"; toggles .Floor1CabPresence
rectangle at (90,370)-(201,411): text "Presence 2"; toggles .Floor2CabPresence
rectangle at (90,470)-(201,511): text "Presence 0"; toggles .Floor0CabPresence
rectangle at (150,690)-(221,751): text "Opened 3"; toggles .Floor3DoorOpened
rectangle at (150,760)-(221,821): text "Opened 2"; toggles .Floor2DoorOpened
rectangle at (150,830)-(221,891): text "Opened 1"; toggles .Floor1DoorOpened
rectangle at (150,900)-(221,961): text "Opened 0"; toggles .Floor0DoorOpened
rectangle at (60,690)-(131,751): text "Closed 3"; toggles .Floor3DoorClosed
rectangle at (60,760)-(131,821): text "Closed 2"; toggles .Floor2DoorClosed
rectangle at (60,830)-(131,891): text "Closed 1"; toggles .Floor1DoorClosed
rectangle at (60,900)-(131,961): text "Closed 0"; toggles .Floor0DoorClosed
rectangle at (90,160)-(201,201): text "INPUTS"
rounded rectangle at (1060,820)-(1151,861): text "Closing 3"; alarm colour if .Floor3DoorClose
rounded rectangle at (1060,870)-(1151,911): text "Closing 2"; alarm colour if .Floor2DoorClose
rounded rectangle at (1060,970)-(1151,1011): text "Closing 0"; alarm colour if .Floor0DoorClose
rounded rectangle at (1060,920)-(1151,961): text "Closing 1"; alarm colour if .Floor1DoorClose
rounded rectangle at (1170,820)-(1261,861): text "Opening 3"; alarm colour if .Floor3DoorOpen
rounded rectangle at (1170,870)-(1261,911): text "Opening 2"; alarm colour if .Floor2DoorOpen
rounded rectangle at (1170,970)-(1261,1011): text "Opening 0"; alarm colour if .Floor0DoorOpen
rounded rectangle at (1170,920)-(1261,961): text "Opening 1"; alarm colour if .Floor1DoorOpen
rectangle at (590,360)-(1001,401): alarm colour if .isBetween[3]
rectangle at (560,260)-(1021,351): text "4"; alarm colour if .Floor[4].CabPresence
rectangle at (560,110)-(1021,201): text "5"; alarm colour if Floor[5].CabPresence
rectangle at (590,210)-(1001,251): alarm colour if .isBetween[4]
ellipse at (610,290)-(641,321): alarm colour if Floor[4].CabLed
ellipse at (610,140)-(641,171): alarm colour if Floor[5].CabLed
rectangle at (740,270)-(811,341): alarm colour if Floor[4].DoorClosed
rectangle at (750,120)-(821,191): alarm colour if Floor[5].DoorClosed
rectangle at (870,270)-(941,341): alarm colour if Floor[4].DoorOpened
rectangle at (870,120)-(941,191): alarm colour if Floor[5].DoorOpened
rectangle at (90,270)-(201,311): text "Presence 4"; toggles .Floor[4].CabPresence
rectangle at (90,220)-(201,261): text "Presence 5"; toggles .Floor[5].CabPresence
rectangle at (150,620)-(221,681): text "Opened 4"; toggles Floor[4].DoorOpened
rectangle at (60,620)-(131,681): text "Closed 4"; toggles Floor[4].DoorClosed
rectangle at (150,550)-(221,611): text "Opened 5"; toggles Floor[5].DoorOpened
rectangle at (60,550)-(131,611): text "Closed 5"; toggles Floor[5].DoorClosed
button at (290,560)-(371,621): text "CallP4"; taps .Cabin.Call[4]
button at (290,490)-(371,551): text "CallP5"; taps .Cabin.Call[5]
rounded rectangle at (1060,770)-(1151,811): text "Closing 4"; alarm colour if .Floor[4].DoorClose
rounded rectangle at (1170,770)-(1261,811): text "Opening 4"; alarm colour if Floor[4].DoorOpen
rounded rectangle at (1060,720)-(1151,761): text "Closing 5"; alarm colour if .Floor[5].DoorClose
rounded rectangle at (1170,720)-(1261,761): text "Opening 5"; alarm colour if .Floor[5].DoorOpen
button at (430,310)-(491,351): text "Down"; taps .Floor[4].CallDw
button at (430,260)-(491,301): text "Up"; taps .Floor[4].CallUp
ellipse at (510,260)-(541,291): alarm colour if Floor[4].LedUp
ellipse at (510,320)-(541,351): alarm colour if Floor[4].LedDw
button at (430,160)-(491,201): text "Down"; taps .Floor[5].CallDw
ellipse at (510,170)-(541,201): alarm colour if Floor[5].LedDw
button at (430,410)-(491,451): text "Up"; taps .Floor[3].CallUp
ellipse at (510,410)-(541,441): alarm colour if Floor[3].LedUp
3 more shapes without text or variables
6 elements of other kinds (tables, trends, ...) not read
*)
